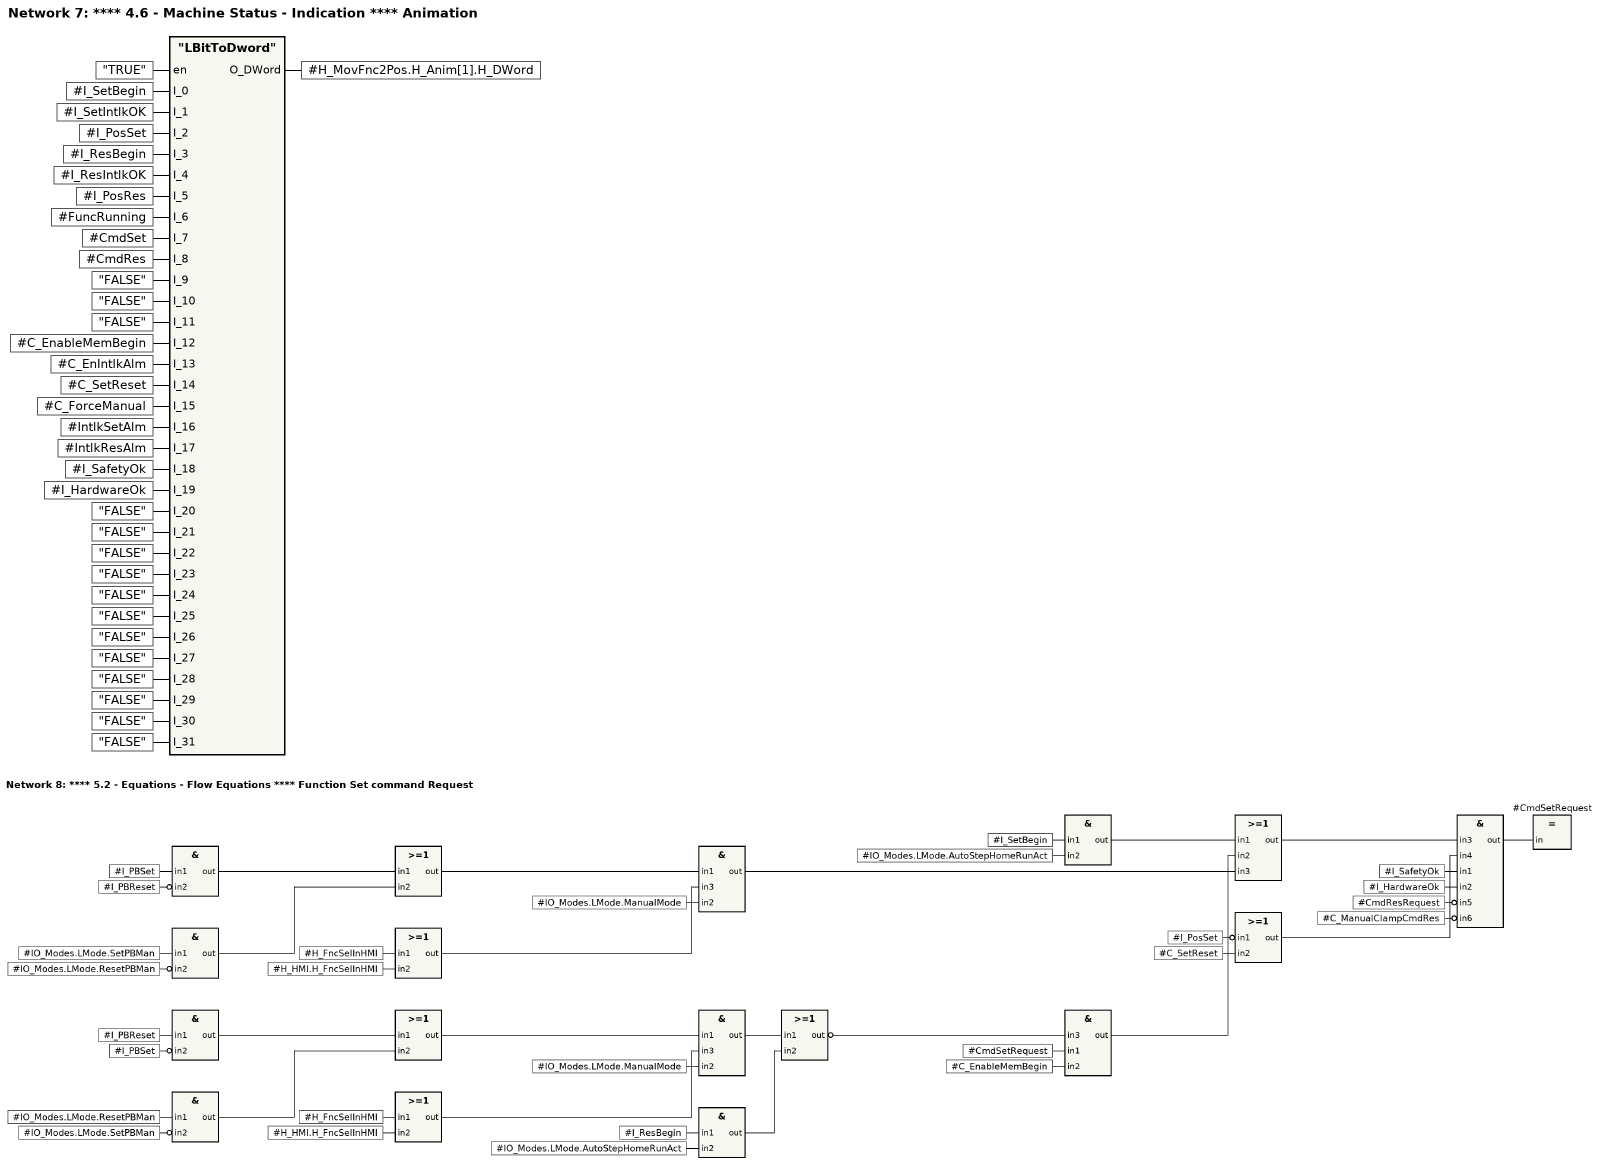
   IF "TRUE" THEN
       "LBitToDword"(I_0 := #I_SetBegin,
                     I_1 := #I_SetIntlkOK,
                     I_2 := #I_PosSet,
                     I_3 := #I_ResBegin,
                     I_4 := #I_ResIntlkOK,
                     I_5 := #I_PosRes,
                     I_6 := #FuncRunning,
                     I_7 := #CmdSet,
                     I_8 := #CmdRes,
                     I_9 := "FALSE",
                     I_10 := "FALSE",
                     I_11 := "FALSE",
                     I_12 := #C_EnableMemBegin,
                     I_13 := #C_EnIntlkAlm,
                     I_14 := #C_SetReset,
                     I_15 := #C_ForceManual,
                     I_16 := #IntlkSetAlm,
                     I_17 := #IntlkResAlm,
                     I_18 := #I_SafetyOk,
                     I_19 := #I_HardwareOk,
                     I_20 := "FALSE",
                     I_21 := "FALSE",
                     I_22 := "FALSE",
                     I_23 := "FALSE",
                     I_24 := "FALSE",
                     I_25 := "FALSE",
                     I_26 := "FALSE",
                     I_27 := "FALSE",
                     I_28 := "FALSE",
                     I_29 := "FALSE",
                     I_30 := "FALSE",
                     I_31 := "FALSE",
                     O_DWord => #H_MovFnc2Pos.H_Anim[1].H_DWord);
   END_IF;
END_REGION

REGION Network 8: **** 5.2 - Equations - Flow Equations **** Function Set command Request
   // Function Set command Request
   #CmdSetRequest := ((#I_SetBegin AND #IO_Modes.LMode.AutoStepHomeRunAct) OR (NOT ((((#I_PBReset AND NOT #I_PBSet) OR (#IO_Modes.LMode.ResetPBMan AND NOT #IO_Modes.LMode.SetPBMan)) AND (#H_FncSelInHMI OR #H_HMI.H_FncSelInHMI) AND #IO_Modes.LMode.ManualMode) OR (#I_ResBegin AND #IO_Modes.LMode.AutoStepHomeRunAct)) AND #CmdSetRequest AND #C_EnableMemBegin) OR (((#I_PBSet AND NOT #I_PBReset) OR (#IO_Modes.LMode.SetPBMan AND NOT #IO_Modes.LMode.ResetPBMan)) AND (#H_FncSelInHMI OR #H_HMI.H_FncSelInHMI) AND #IO_Modes.LMode.ManualMode)) AND (NOT #I_PosSet OR #C_SetReset) AND #I_SafetyOk AND #I_HardwareOk AND NOT #CmdResRequest AND NOT #C_ManualClampCmdRes;
END_REGION

REGION Network 9: **** 5.2 - Equations - Flow Equations **** Function Reset command Request
   // Function Reset command Request
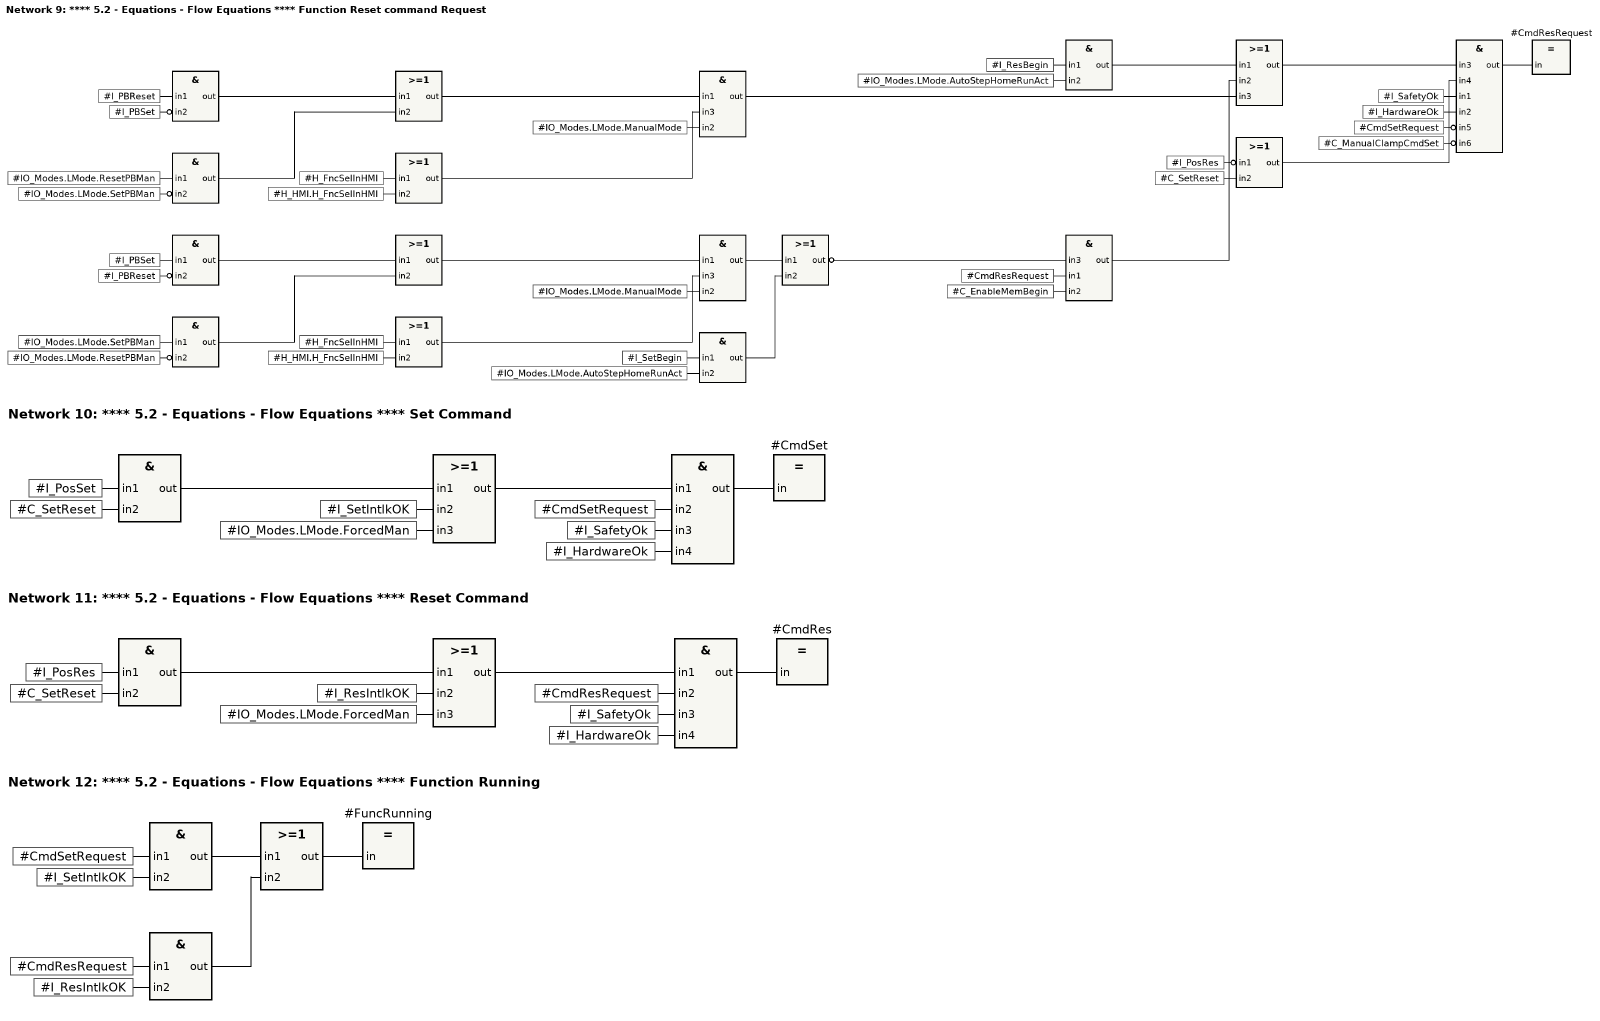
   #CmdResRequest := ((#I_ResBegin AND #IO_Modes.LMode.AutoStepHomeRunAct) OR (NOT ((((#I_PBSet AND NOT #I_PBReset) OR (#IO_Modes.LMode.SetPBMan AND NOT #IO_Modes.LMode.ResetPBMan)) AND (#H_FncSelInHMI OR #H_HMI.H_FncSelInHMI) AND #IO_Modes.LMode.ManualMode) OR (#I_SetBegin AND #IO_Modes.LMode.AutoStepHomeRunAct)) AND #CmdResRequest AND #C_EnableMemBegin) OR (((#I_PBReset AND NOT #I_PBSet) OR (#IO_Modes.LMode.ResetPBMan AND NOT #IO_Modes.LMode.SetPBMan)) AND (#H_FncSelInHMI OR #H_HMI.H_FncSelInHMI) AND #IO_Modes.LMode.ManualMode)) AND (NOT #I_PosRes OR #C_SetReset) AND #I_SafetyOk AND #I_HardwareOk AND NOT #CmdSetRequest AND NOT #C_ManualClampCmdSet;
END_REGION

REGION Network 10: **** 5.2 - Equations - Flow Equations **** Set Command
   // Set Command
   #CmdSet := ((#I_PosSet AND #C_SetReset) OR #I_SetIntlkOK OR #IO_Modes.LMode.ForcedMan) AND #CmdSetRequest AND #I_SafetyOk AND #I_HardwareOk;
END_REGION

REGION Network 11: **** 5.2 - Equations - Flow Equations **** Reset Command
   // Reset Command
   #CmdRes := ((#I_PosRes AND #C_SetReset) OR #I_ResIntlkOK OR #IO_Modes.LMode.ForcedMan) AND #CmdResRequest AND #I_SafetyOk AND #I_HardwareOk;
END_REGION

REGION Network 12: **** 5.2 - Equations - Flow Equations **** Function Running
   // Function Running
   #FuncRunning := (#CmdSetRequest AND #I_SetIntlkOK) OR (#CmdResRequest AND #I_ResIntlkOK);
END_REGION

REGION Network 13: **** 5.2 - Equations - Flow Equations **** Function Running Memory
   // Function Running Memory
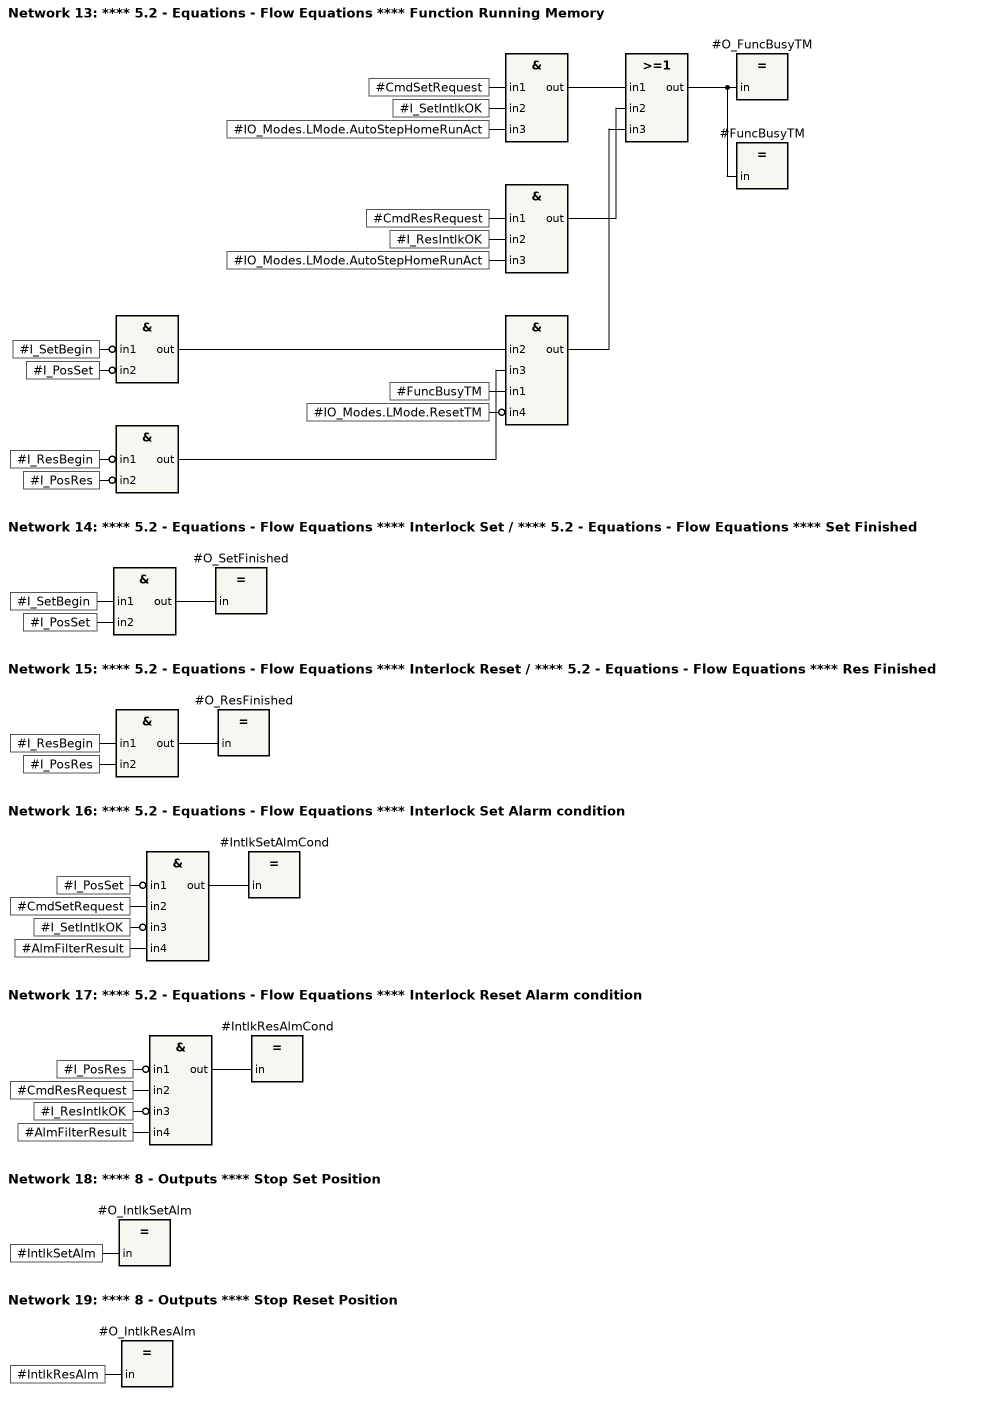
   #O_FuncBusyTM := (#CmdSetRequest AND #I_SetIntlkOK AND #IO_Modes.LMode.AutoStepHomeRunAct) OR (#CmdResRequest AND #I_ResIntlkOK AND #IO_Modes.LMode.AutoStepHomeRunAct) OR (NOT #I_SetBegin AND NOT #I_PosSet AND NOT #I_ResBegin AND NOT #I_PosRes AND #FuncBusyTM AND NOT #IO_Modes.LMode.ResetTM);
   #FuncBusyTM := #O_FuncBusyTM;
END_REGION

REGION Network 14: **** 5.2 - Equations - Flow Equations **** Interlock Set / **** 5.2 - Equations - Flow Equations **** Set Finished
   // Interlock Set
   #O_SetFinished := #I_SetBegin AND #I_PosSet;
END_REGION

REGION Network 15: **** 5.2 - Equations - Flow Equations **** Interlock Reset / **** 5.2 - Equations - Flow Equations **** Res Finished
   // Interlock Reset
   #O_ResFinished := #I_ResBegin AND #I_PosRes;
END_REGION

REGION Network 16: **** 5.2 - Equations - Flow Equations **** Interlock Set Alarm condition
   // Interlock Set Alarm condition
   #IntlkSetAlmCond := NOT #I_PosSet AND #CmdSetRequest AND NOT #I_SetIntlkOK AND #AlmFilterResult;
END_REGION

REGION Network 17: **** 5.2 - Equations - Flow Equations **** Interlock Reset Alarm condition
   // Interlock Reset Alarm condition
   #IntlkResAlmCond := NOT #I_PosRes AND #CmdResRequest AND NOT #I_ResIntlkOK AND #AlmFilterResult;
END_REGION

REGION Network 18: **** 8 - Outputs **** Stop Set Position
   // Stop Set Position
   #O_IntlkSetAlm := #IntlkSetAlm;
END_REGION

REGION Network 19: **** 8 - Outputs **** Stop Reset Position
   // Stop Reset Position
   #O_IntlkResAlm := #IntlkResAlm;
END_REGION

REGION Network 20: **** 8 - Outputs **** Function is Selected in manual Mode
   // Function is Selected in manual Mode
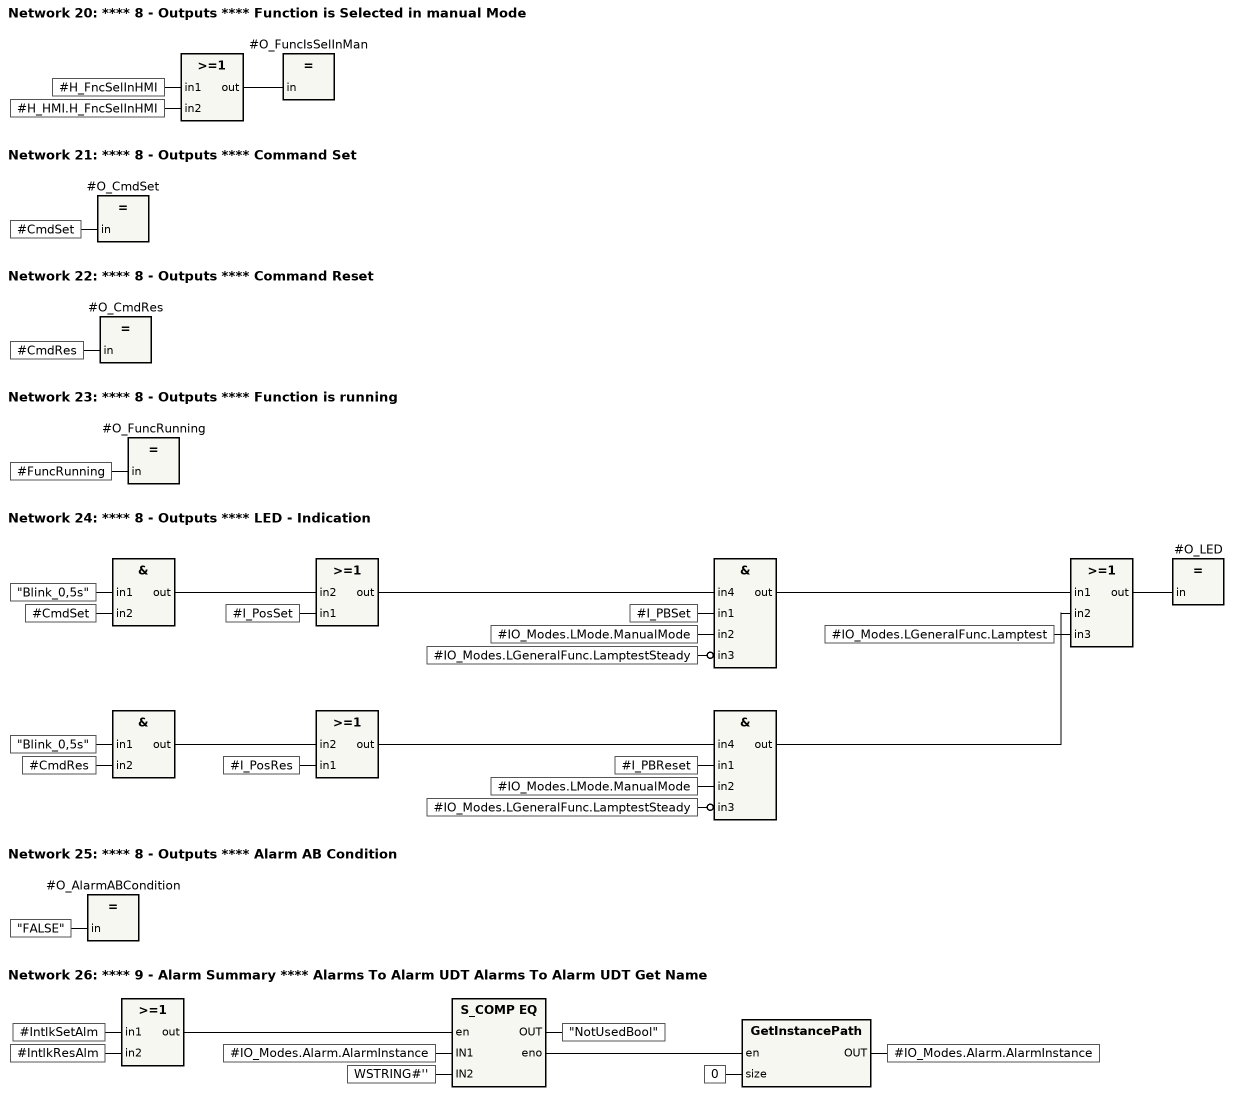
   #O_FuncIsSelInMan := #H_FncSelInHMI OR #H_HMI.H_FncSelInHMI;
END_REGION

REGION Network 21: **** 8 - Outputs **** Command Set
   // Command set
   #O_CmdSet := #CmdSet;
END_REGION

REGION Network 22: **** 8 - Outputs **** Command Reset
   // Command Reset
   #O_CmdRes := #CmdRes;
END_REGION

REGION Network 23: **** 8 - Outputs **** Function is running
   // Function is running
   #O_FuncRunning := #FuncRunning;
END_REGION

REGION Network 24: **** 8 - Outputs **** LED - Indication
   // LED - Indication
   #O_LED := ((("Blink_0,5s" AND #CmdSet) OR #I_PosSet) AND #I_PBSet AND #IO_Modes.LMode.ManualMode AND NOT #IO_Modes.LGeneralFunc.LamptestSteady) OR ((("Blink_0,5s" AND #CmdRes) OR #I_PosRes) AND #I_PBReset AND #IO_Modes.LMode.ManualMode AND NOT #IO_Modes.LGeneralFunc.LamptestSteady) OR #IO_Modes.LGeneralFunc.Lamptest;
END_REGION

REGION Network 25: **** 8 - Outputs **** Alarm AB Condition
   // Alarm AB Condition
   #O_AlarmABCondition := "FALSE";
END_REGION

REGION Network 26: **** 9 - Alarm Summary **** Alarms To Alarm UDT Alarms To Alarm UDT Get Name
   // Alarm / Alarm D
   S_COMP(EN := #IntlkSetAlm OR #IntlkResAlm,
          IN1 := #IO_Modes.Alarm.AlarmInstance,
          IN2 := WSTRING#'',
          OUT => "NotUsedBool",
          ENO => #_w1);
   IF #_w1 THEN GetInstancePath(size := 0, OUT => #IO_Modes.Alarm.AlarmInstance); END_IF;
END_REGION

REGION Network 27: **** 9 - Alarm Summary **** Alarms To Alarm UDT
   // Alarm / Alarm D
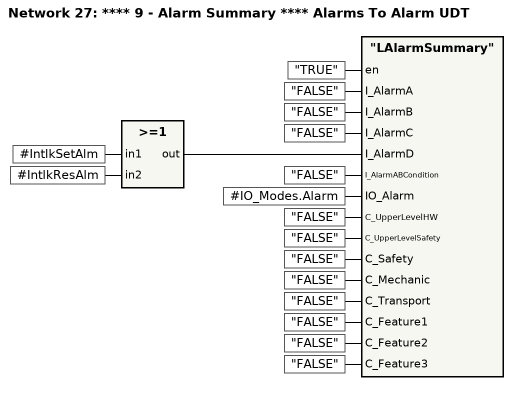
   IF "TRUE" THEN
       "LAlarmSummary"(I_AlarmA := "FALSE",
                       I_AlarmB := "FALSE",
                       I_AlarmC := "FALSE",
                       I_AlarmD := #IntlkSetAlm OR #IntlkResAlm,
                       I_AlarmABCondition := "FALSE",
                       IO_Alarm := #IO_Modes.Alarm,
                       C_UpperLevelHW := "FALSE",
                       C_UpperLevelSafety := "FALSE",
                       C_Safety := "FALSE",
                       C_Mechanic := "FALSE",
                       C_Transport := "FALSE",
                       C_Feature1 := "FALSE",
                       C_Feature2 := "FALSE",
                       C_Feature3 := "FALSE");
   END_IF;
END_REGION
END_FUNCTION_BLOCK

FUNCTION_BLOCK "LGeneralReverse"   // FB1103, FBD
TITLE = LGeneralReverse
{ S7_Optimized_Access := 'TRUE' }
VERSION : 0.1
// stored: AutoNumber false, IsIECCheckEnabled false, IsRetainMemResEnabled false, MemoryReserve 100, SetENOAutomatically False, UDAEnableTagReadback false
   VAR_INPUT
      I_GeneralReverseSw { ExternalAccessible := 'False'; ExternalVisible := 'False'; ExternalWritable := 'False'} : Bool;   // General reverse switch
      I_FbkContactorFwd { ExternalAccessible := 'False'; ExternalVisible := 'False'; ExternalWritable := 'False'} : Bool;   // Feedback contactor Forward
      I_FbkContactorBwd { ExternalAccessible := 'False'; ExternalVisible := 'False'; ExternalWritable := 'False'} : Bool;   // Feedback contactor Backward
      I_EnableAlarm { ExternalAccessible := 'False'; ExternalVisible := 'False'; ExternalWritable := 'False'} : Bool;   // Enable alarm / Enable Alarm
      I_ResetFbkAlarm { ExternalAccessible := 'False'; ExternalVisible := 'False'; ExternalWritable := 'False'} : Bool;   // Reset feedback alarm / Alarm reset pushbutton is activated
      C_FeedbackUsed { ExternalAccessible := 'False'; ExternalVisible := 'False'; ExternalWritable := 'False'} : Bool;   // Config Feedback used
   END_VAR
   VAR_OUTPUT
      O_ContactorFwd { ExternalAccessible := 'False'; ExternalVisible := 'False'; ExternalWritable := 'False'} : Bool;   // Activate low speed contactor / Activate Forward contactor
      O_ContactorBwd { ExternalAccessible := 'False'; ExternalVisible := 'False'; ExternalWritable := 'False'} : Bool;   // Activate High Speed contactor / Activate Backward contactor
      O_GenRevSw { ExternalAccessible := 'False'; ExternalVisible := 'False'; ExternalWritable := 'False'} : Bool;   // General reverse switch
      O_AlarmABCondition { ExternalAccessible := 'False'; ExternalVisible := 'False'; ExternalWritable := 'False'} : Bool;   // Alarm AB Condition
      O_AlarmA { ExternalAccessible := 'False'; ExternalVisible := 'False'; ExternalWritable := 'False'} : Bool;   // Alarm A
      O_AlarmB { ExternalAccessible := 'False'; ExternalVisible := 'False'; ExternalWritable := 'False'} : Bool;   // Alarm B
      O_AlarmC { ExternalAccessible := 'False'; ExternalVisible := 'False'; ExternalWritable := 'False'} : Bool;   // Alarm C
      O_AlarmD { ExternalAccessible := 'False'; ExternalVisible := 'False'; ExternalWritable := 'False'} : Bool;   // Alarm D
      H_AlarmDWord { ExternalAccessible := 'False'; ExternalVisible := 'False'; ExternalWritable := 'False'} : DWord;   // Alarm Word
   END_VAR
   VAR_IN_OUT
      IO_Modes : "Modes";   // Modes
      H_HMI : "H_HMI";   // Icon Animation
      H_GeneralReverse : "H_GeneralReverse";   // Animation
   END_VAR
   VAR
      AB_FbkContactorFwd { ExternalAccessible := 'False'; ExternalVisible := 'False'; ExternalWritable := 'False'} : Bool;   // Feedback error Contactor Forward
      AB_FbkContactorBwd { ExternalAccessible := 'False'; ExternalVisible := 'False'; ExternalWritable := 'False'} : Bool;   // Feedback error Contactor Backward
      AB_GeneralReverseSw { ExternalAccessible := 'False'; ExternalVisible := 'False'; ExternalWritable := 'False'} : Bool;   // General reverse is activated
      AC_GeneralReverseSw { ExternalAccessible := 'False'; ExternalVisible := 'False'; ExternalWritable := 'False'} : Bool;   // General reverse Switch is active
      FbkContactorFwdAlmCond { ExternalAccessible := 'False'; ExternalVisible := 'False'; ExternalWritable := 'False'} : Bool;   // Motor protection alarm condition / Motor protection Alarm condition / Feedback Contactor Forward Alarm condition
      FbkContactorBwdAlmCond { ExternalAccessible := 'False'; ExternalVisible := 'False'; ExternalWritable := 'False'} : Bool;   // Motor protection alarm condition / Motor protection Alarm condition / Feedback Contactor Backward Alarm condition
      AlarmA { ExternalAccessible := 'False'; ExternalVisible := 'False'; ExternalWritable := 'False'} : Bool;   // Alarm A
      AlarmB { ExternalAccessible := 'False'; ExternalVisible := 'False'; ExternalWritable := 'False'} : Bool;   // Alarm B
      AlarmC { ExternalAccessible := 'False'; ExternalVisible := 'False'; ExternalWritable := 'False'} : Bool;   // Alarm C
      AlarmD { ExternalAccessible := 'False'; ExternalVisible := 'False'; ExternalWritable := 'False'} : Bool;   // Alarm D
      AlarmABCondition { ExternalAccessible := 'False'; ExternalVisible := 'False'; ExternalWritable := 'False'} : Bool;   // Alarm AB Condition
      ContactorFwd { ExternalAccessible := 'False'; ExternalVisible := 'False'; ExternalWritable := 'False'} : Bool;   // Activate low speed contactor / Activate Forward contactor
      ContactorBwd { ExternalAccessible := 'False'; ExternalVisible := 'False'; ExternalWritable := 'False'} : Bool;   // Activate High Speed contactor / Activate Backward contactor
      _TimerInit { ExternalAccessible := 'False'; ExternalVisible := 'False'; ExternalWritable := 'False'} : TON_TIME;   // Timer
      _TimerContactorFwd { ExternalAccessible := 'False'; ExternalVisible := 'False'; ExternalWritable := 'False'} : TON_TIME;   // Timer
      _TimerContactorBwd { ExternalAccessible := 'False'; ExternalVisible := 'False'; ExternalWritable := 'False'} : TON_TIME;   // Timer
      _TimerContactorFwdFbk { ExternalAccessible := 'False'; ExternalVisible := 'False'; ExternalWritable := 'False'} : TON_TIME;   // Timer
      _TimerContactorBwdFbk { ExternalAccessible := 'False'; ExternalVisible := 'False'; ExternalWritable := 'False'} : TON_TIME;   // Timer
      _ContactorFwdFbk { ExternalAccessible := 'False'; ExternalVisible := 'False'; ExternalWritable := 'False'} : "L1AlarmMultiIn";   // FB
      _ContactorBwdFbk { ExternalAccessible := 'False'; ExternalVisible := 'False'; ExternalWritable := 'False'} : "L1AlarmMultiIn";   // FB
      Edge { ExternalAccessible := 'False'; ExternalVisible := 'False'; ExternalWritable := 'False'} : Array[1..10] of Bool;   // Edge
   END_VAR
   VAR_TEMP   // added for the SCL form of the ladder/FBD networks
      _w1 : Bool;
      _w2 : Bool;
   END_VAR
BEGIN

REGION Network 1: ****2.1 - Enable Alarms **** Enable Contactor Forward Feedback Alarm
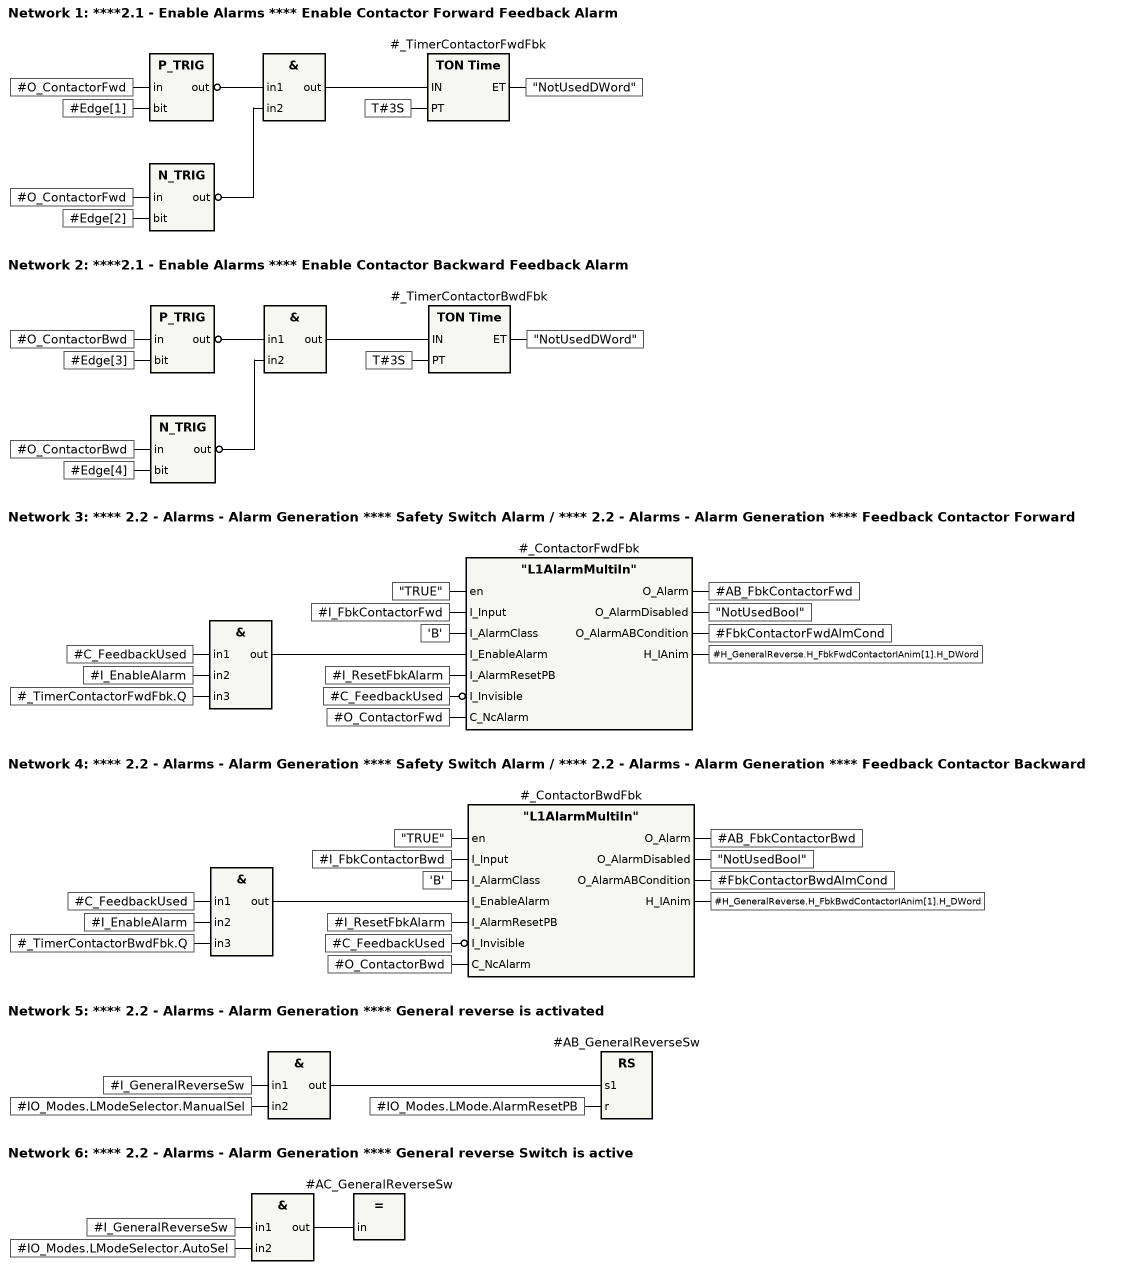
   #_w1 := #O_ContactorFwd AND NOT #Edge[1];   // rising edge
   #Edge[1] := #O_ContactorFwd;
   #_w2 := NOT #O_ContactorFwd AND #Edge[2];   // falling edge
   #Edge[2] := #O_ContactorFwd;
   #_TimerContactorFwdFbk(IN := NOT #_w1 AND NOT #_w2, PT := T#3S, ET => "NotUsedDWord");   // TON
END_REGION

REGION Network 2: ****2.1 - Enable Alarms **** Enable Contactor Backward Feedback Alarm
   #_w1 := #O_ContactorBwd AND NOT #Edge[3];   // rising edge
   #Edge[3] := #O_ContactorBwd;
   #_w2 := NOT #O_ContactorBwd AND #Edge[4];   // falling edge
   #Edge[4] := #O_ContactorBwd;
   #_TimerContactorBwdFbk(IN := NOT #_w1 AND NOT #_w2, PT := T#3S, ET => "NotUsedDWord");   // TON
END_REGION

REGION Network 3: **** 2.2 - Alarms - Alarm Generation **** Safety Switch Alarm / **** 2.2 - Alarms - Alarm Generation **** Feedback Contactor Forward
   // Safety Switch Alarm / Feedback error Contactor Forward
   IF "TRUE" THEN
       #_ContactorFwdFbk(I_Input := #I_FbkContactorFwd,   // "L1AlarmMultiIn"
                         I_AlarmClass := 'B',
                         I_EnableAlarm := #C_FeedbackUsed AND #I_EnableAlarm AND #_TimerContactorFwdFbk.Q,
                         I_AlarmResetPB := #I_ResetFbkAlarm,
                         I_Invisible := NOT #C_FeedbackUsed,
                         C_NcAlarm := #O_ContactorFwd,
                         O_Alarm => #AB_FbkContactorFwd,
                         O_AlarmDisabled => "NotUsedBool",
                         O_AlarmABCondition => #FbkContactorFwdAlmCond,
                         H_IAnim => #H_GeneralReverse.H_FbkFwdContactorIAnim[1].H_DWord);
   END_IF;
END_REGION

REGION Network 4: **** 2.2 - Alarms - Alarm Generation **** Safety Switch Alarm / **** 2.2 - Alarms - Alarm Generation **** Feedback Contactor Backward
   // Safety Switch Alarm / Feedback error Contactor Backward
   IF "TRUE" THEN
       #_ContactorBwdFbk(I_Input := #I_FbkContactorBwd,   // "L1AlarmMultiIn"
                         I_AlarmClass := 'B',
                         I_EnableAlarm := #C_FeedbackUsed AND #I_EnableAlarm AND #_TimerContactorBwdFbk.Q,
                         I_AlarmResetPB := #I_ResetFbkAlarm,
                         I_Invisible := NOT #C_FeedbackUsed,
                         C_NcAlarm := #O_ContactorBwd,
                         O_Alarm => #AB_FbkContactorBwd,
                         O_AlarmDisabled => "NotUsedBool",
                         O_AlarmABCondition => #FbkContactorBwdAlmCond,
                         H_IAnim => #H_GeneralReverse.H_FbkBwdContactorIAnim[1].H_DWord);
   END_IF;
END_REGION

REGION Network 5: **** 2.2 - Alarms - Alarm Generation **** General reverse is activated
   IF #IO_Modes.LMode.AlarmResetPB THEN
       #AB_GeneralReverseSw := FALSE;   // RS flip-flop
   END_IF;
   IF #I_GeneralReverseSw AND #IO_Modes.LModeSelector.ManualSel THEN #AB_GeneralReverseSw := TRUE; END_IF;
END_REGION

REGION Network 6: **** 2.2 - Alarms - Alarm Generation **** General reverse Switch is active
   #AC_GeneralReverseSw := #I_GeneralReverseSw AND #IO_Modes.LModeSelector.AutoSel;
END_REGION

REGION Network 7: **** 4.6 - Machine Status - Indication **** Low Speed Contactor Animation / **** 4.6 - Machine Status - Indication **** Forward Contactor Animation
   // Low speed Contactor Animation
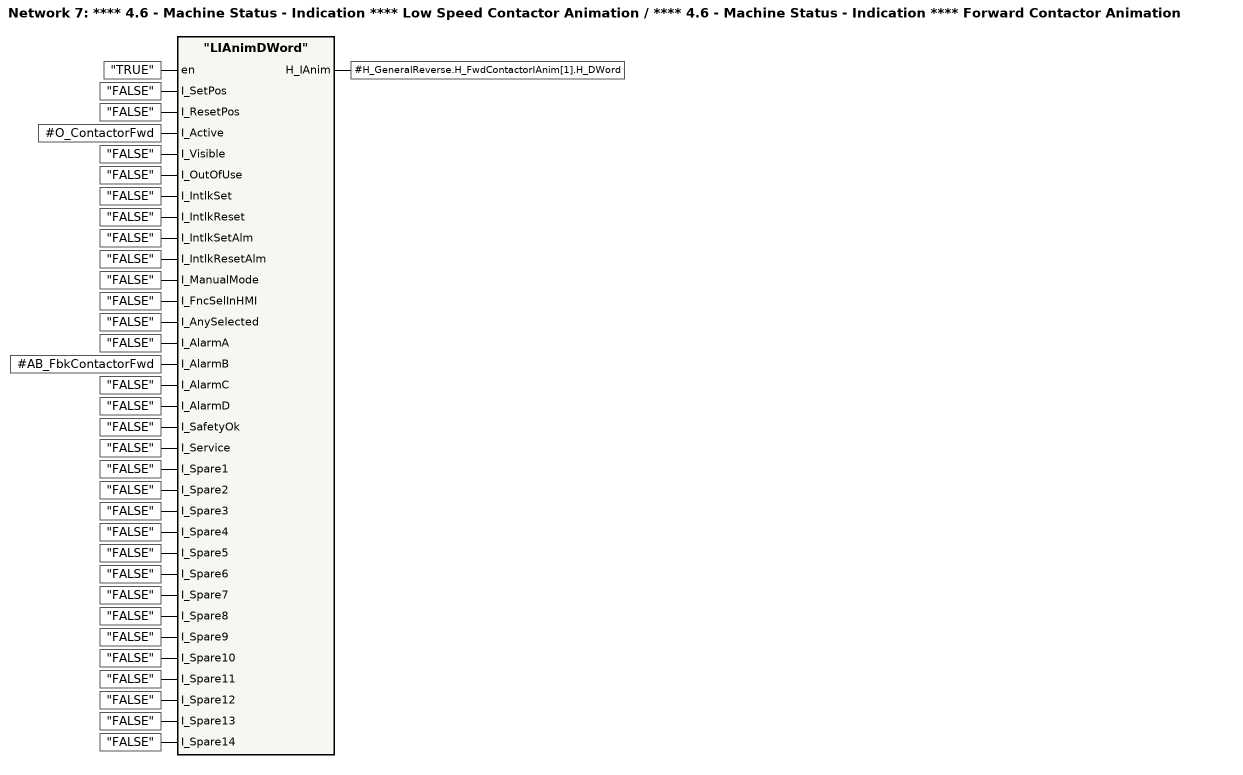
   IF "TRUE" THEN
       "LIAnimDWord"(I_SetPos := "FALSE",
                     I_ResetPos := "FALSE",
                     I_Active := #O_ContactorFwd,
                     I_Visible := "FALSE",
                     I_OutOfUse := "FALSE",
                     I_IntlkSet := "FALSE",
                     I_IntlkReset := "FALSE",
                     I_IntlkSetAlm := "FALSE",
                     I_IntlkResetAlm := "FALSE",
                     I_ManualMode := "FALSE",
                     I_FncSelInHMI := "FALSE",
                     I_AnySelected := "FALSE",
                     I_AlarmA := "FALSE",
                     I_AlarmB := #AB_FbkContactorFwd,
                     I_AlarmC := "FALSE",
                     I_AlarmD := "FALSE",
                     I_SafetyOk := "FALSE",
                     I_Service := "FALSE",
                     I_Spare1 := "FALSE",
                     I_Spare2 := "FALSE",
                     I_Spare3 := "FALSE",
                     I_Spare4 := "FALSE",
                     I_Spare5 := "FALSE",
                     I_Spare6 := "FALSE",
                     I_Spare7 := "FALSE",
                     I_Spare8 := "FALSE",
                     I_Spare9 := "FALSE",
                     I_Spare10 := "FALSE",
                     I_Spare11 := "FALSE",
                     I_Spare12 := "FALSE",
                     I_Spare13 := "FALSE",
                     I_Spare14 := "FALSE",
                     H_IAnim => #H_GeneralReverse.H_FwdContactorIAnim[1].H_DWord);
   END_IF;
END_REGION

REGION Network 8: **** 4.6 - Machine Status - Indication **** High Speed Contactor Animation / **** 4.6 - Machine Status - Indication **** Backward Contactor Animation
   // High Speed Contactor Animation
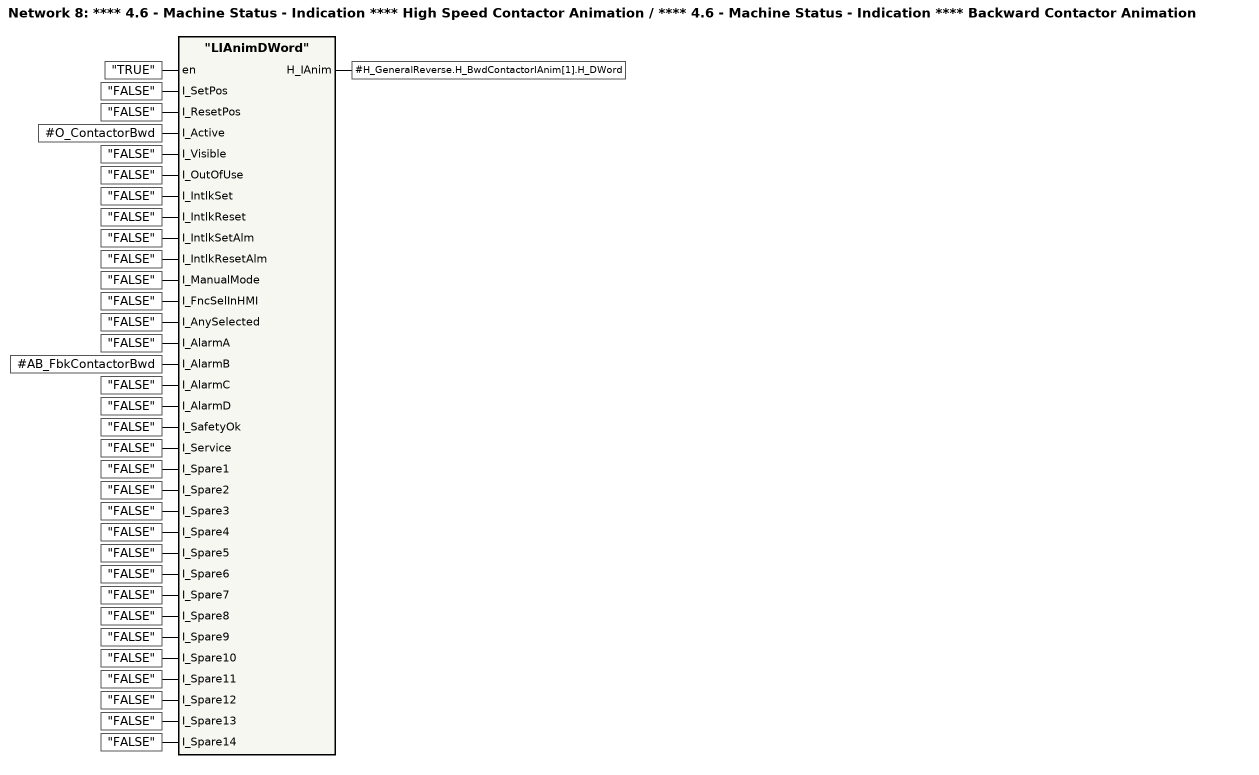
   IF "TRUE" THEN
       "LIAnimDWord"(I_SetPos := "FALSE",
                     I_ResetPos := "FALSE",
                     I_Active := #O_ContactorBwd,
                     I_Visible := "FALSE",
                     I_OutOfUse := "FALSE",
                     I_IntlkSet := "FALSE",
                     I_IntlkReset := "FALSE",
                     I_IntlkSetAlm := "FALSE",
                     I_IntlkResetAlm := "FALSE",
                     I_ManualMode := "FALSE",
                     I_FncSelInHMI := "FALSE",
                     I_AnySelected := "FALSE",
                     I_AlarmA := "FALSE",
                     I_AlarmB := #AB_FbkContactorBwd,
                     I_AlarmC := "FALSE",
                     I_AlarmD := "FALSE",
                     I_SafetyOk := "FALSE",
                     I_Service := "FALSE",
                     I_Spare1 := "FALSE",
                     I_Spare2 := "FALSE",
                     I_Spare3 := "FALSE",
                     I_Spare4 := "FALSE",
                     I_Spare5 := "FALSE",
                     I_Spare6 := "FALSE",
                     I_Spare7 := "FALSE",
                     I_Spare8 := "FALSE",
                     I_Spare9 := "FALSE",
                     I_Spare10 := "FALSE",
                     I_Spare11 := "FALSE",
                     I_Spare12 := "FALSE",
                     I_Spare13 := "FALSE",
                     I_Spare14 := "FALSE",
                     H_IAnim => #H_GeneralReverse.H_BwdContactorIAnim[1].H_DWord);
   END_IF;
END_REGION

REGION Network 9: **** 4.6 - Machine Status - Indication **** Stop Detection Reset / **** 4.6 - Machine Status - Indications **** General Reverse Switch Animation
   // Stop Detection Reset
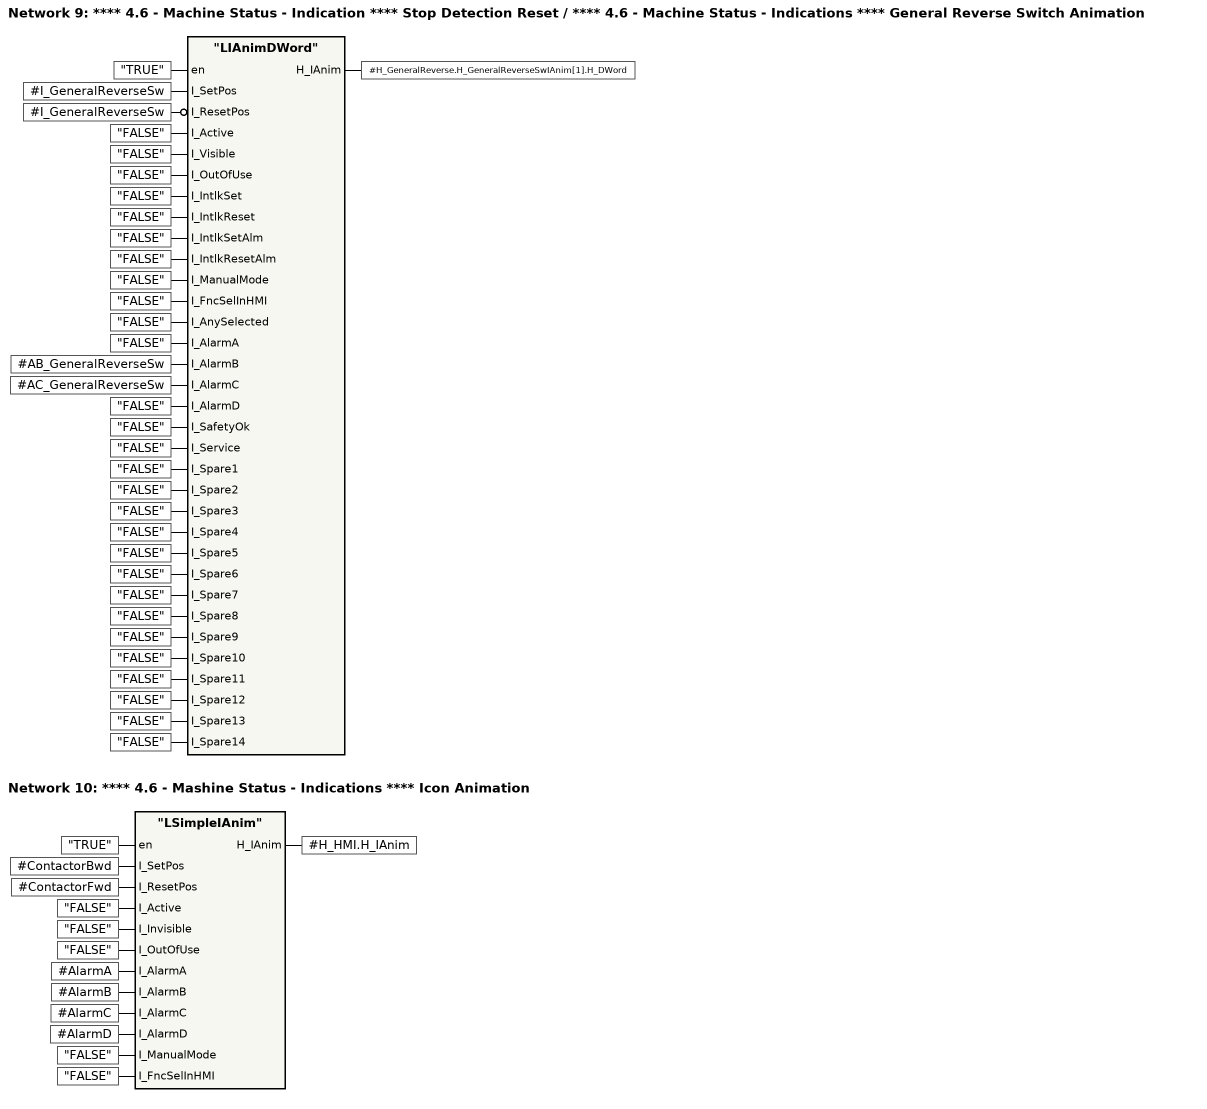
   IF "TRUE" THEN
       "LIAnimDWord"(I_SetPos := #I_GeneralReverseSw,
                     I_ResetPos := NOT #I_GeneralReverseSw,
                     I_Active := "FALSE",
                     I_Visible := "FALSE",
                     I_OutOfUse := "FALSE",
                     I_IntlkSet := "FALSE",
                     I_IntlkReset := "FALSE",
                     I_IntlkSetAlm := "FALSE",
                     I_IntlkResetAlm := "FALSE",
                     I_ManualMode := "FALSE",
                     I_FncSelInHMI := "FALSE",
                     I_AnySelected := "FALSE",
                     I_AlarmA := "FALSE",
                     I_AlarmB := #AB_GeneralReverseSw,
                     I_AlarmC := #AC_GeneralReverseSw,
                     I_AlarmD := "FALSE",
                     I_SafetyOk := "FALSE",
                     I_Service := "FALSE",
                     I_Spare1 := "FALSE",
                     I_Spare2 := "FALSE",
                     I_Spare3 := "FALSE",
                     I_Spare4 := "FALSE",
                     I_Spare5 := "FALSE",
                     I_Spare6 := "FALSE",
                     I_Spare7 := "FALSE",
                     I_Spare8 := "FALSE",
                     I_Spare9 := "FALSE",
                     I_Spare10 := "FALSE",
                     I_Spare11 := "FALSE",
                     I_Spare12 := "FALSE",
                     I_Spare13 := "FALSE",
                     I_Spare14 := "FALSE",
                     H_IAnim => #H_GeneralReverse.H_GeneralReverseSwIAnim[1].H_DWord);
   END_IF;
END_REGION

REGION Network 10: **** 4.6 - Mashine Status - Indications **** Icon Animation
   // Icon Animation
   IF "TRUE" THEN
       "LSimpleIAnim"(I_SetPos := #ContactorBwd,
                      I_ResetPos := #ContactorFwd,
                      I_Active := "FALSE",
                      I_Invisible := "FALSE",
                      I_OutOfUse := "FALSE",
                      I_AlarmA := #AlarmA,
                      I_AlarmB := #AlarmB,
                      I_AlarmC := #AlarmC,
                      I_AlarmD := #AlarmD,
                      I_ManualMode := "FALSE",
                      I_FncSelInHMI := "FALSE",
                      H_IAnim => #H_HMI.H_IAnim);
   END_IF;
END_REGION

REGION Network 11: **** 4.6 - Machine status - Indications **** Animation
   // Animation Word 1
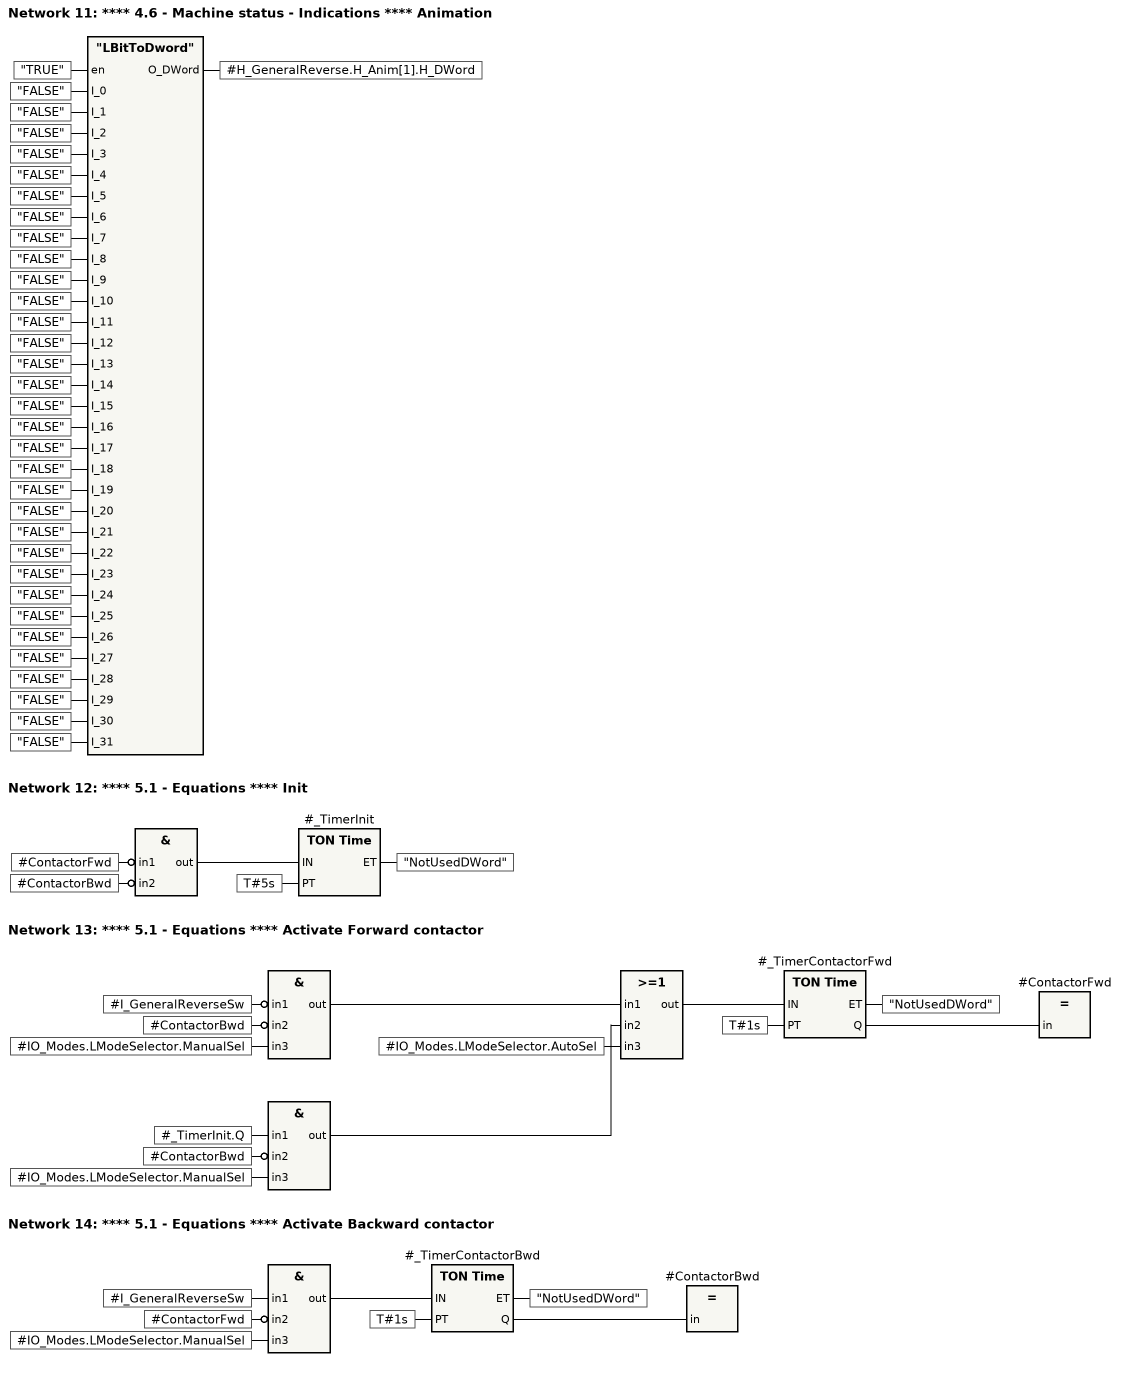
   IF "TRUE" THEN
       "LBitToDword"(I_0 := "FALSE",
                     I_1 := "FALSE",
                     I_2 := "FALSE",
                     I_3 := "FALSE",
                     I_4 := "FALSE",
                     I_5 := "FALSE",
                     I_6 := "FALSE",
                     I_7 := "FALSE",
                     I_8 := "FALSE",
                     I_9 := "FALSE",
                     I_10 := "FALSE",
                     I_11 := "FALSE",
                     I_12 := "FALSE",
                     I_13 := "FALSE",
                     I_14 := "FALSE",
                     I_15 := "FALSE",
                     I_16 := "FALSE",
                     I_17 := "FALSE",
                     I_18 := "FALSE",
                     I_19 := "FALSE",
                     I_20 := "FALSE",
                     I_21 := "FALSE",
                     I_22 := "FALSE",
                     I_23 := "FALSE",
                     I_24 := "FALSE",
                     I_25 := "FALSE",
                     I_26 := "FALSE",
                     I_27 := "FALSE",
                     I_28 := "FALSE",
                     I_29 := "FALSE",
                     I_30 := "FALSE",
                     I_31 := "FALSE",
                     O_DWord => #H_GeneralReverse.H_Anim[1].H_DWord);
   END_IF;
END_REGION

REGION Network 12: **** 5.1 - Equations **** Init
   #_TimerInit(IN := NOT #ContactorFwd AND NOT #ContactorBwd, PT := T#5s, ET => "NotUsedDWord");   // TON
END_REGION

REGION Network 13: **** 5.1 - Equations **** Activate Forward contactor
   #_TimerContactorFwd(IN := (NOT #I_GeneralReverseSw AND NOT #ContactorBwd AND #IO_Modes.LModeSelector.ManualSel) OR (#_TimerInit.Q AND NOT #ContactorBwd AND #IO_Modes.LModeSelector.ManualSel) OR #IO_Modes.LModeSelector.AutoSel,   // TON
                       PT := T#1s,
                       ET => "NotUsedDWord");
   #ContactorFwd := #_TimerContactorFwd.Q;
END_REGION

REGION Network 14: **** 5.1 - Equations **** Activate Backward contactor
   #_TimerContactorBwd(IN := #I_GeneralReverseSw AND NOT #ContactorFwd AND #IO_Modes.LModeSelector.ManualSel,   // TON
                       PT := T#1s,
                       ET => "NotUsedDWord");
   #ContactorBwd := #_TimerContactorBwd.Q;
END_REGION

REGION Network 15: **** 8 - Outputs **** Alarm AB Condition
   // Alarm AB Condition
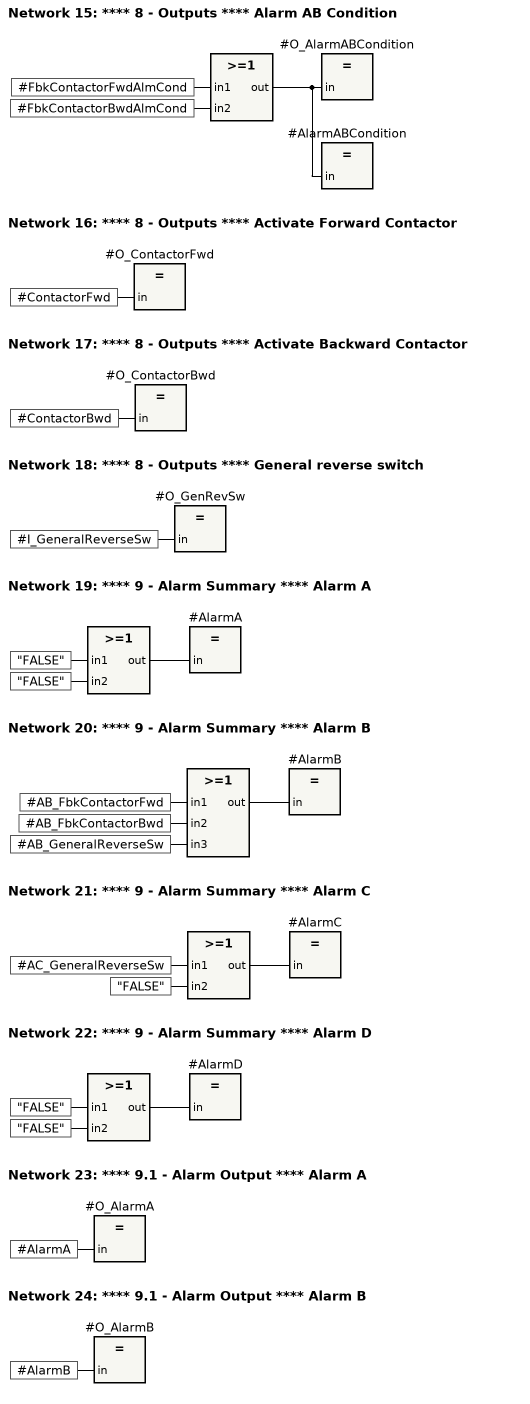
   #O_AlarmABCondition := #FbkContactorFwdAlmCond OR #FbkContactorBwdAlmCond;
   #AlarmABCondition := #O_AlarmABCondition;
END_REGION

REGION Network 16: **** 8 - Outputs **** Activate Forward Contactor
   #O_ContactorFwd := #ContactorFwd;
END_REGION

REGION Network 17: **** 8 - Outputs **** Activate Backward Contactor
   #O_ContactorBwd := #ContactorBwd;
END_REGION

REGION Network 18: **** 8 - Outputs **** General reverse switch
   #O_GenRevSw := #I_GeneralReverseSw;
END_REGION

REGION Network 19: **** 9 - Alarm Summary **** Alarm A
   // Alarm A
   #AlarmA := "FALSE" OR "FALSE";
END_REGION

REGION Network 20: **** 9 - Alarm Summary **** Alarm B
   // Alarm B
   #AlarmB := #AB_FbkContactorFwd OR #AB_FbkContactorBwd OR #AB_GeneralReverseSw;
END_REGION

REGION Network 21: **** 9 - Alarm Summary **** Alarm C
   // Alarm C
   #AlarmC := #AC_GeneralReverseSw OR "FALSE";
END_REGION

REGION Network 22: **** 9 - Alarm Summary **** Alarm D
   // Alarm D
   #AlarmD := "FALSE" OR "FALSE";
END_REGION

REGION Network 23: **** 9.1 - Alarm Output **** Alarm A
   // Alarm A
   #O_AlarmA := #AlarmA;
END_REGION

REGION Network 24: **** 9.1 - Alarm Output **** Alarm B
   // Alarm B
   #O_AlarmB := #AlarmB;
END_REGION

REGION Network 25: **** 9.1 - Alarm Output **** Alarm C
   // Alarm C
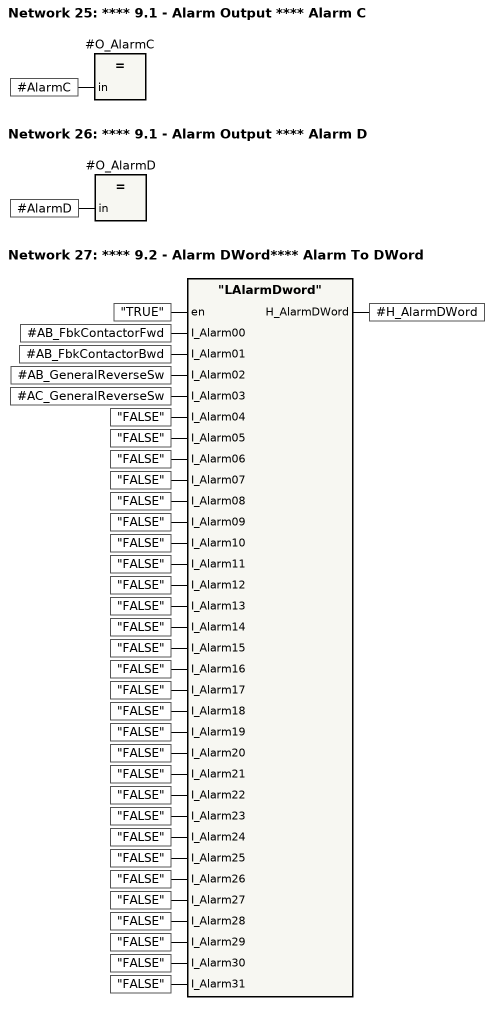
   #O_AlarmC := #AlarmC;
END_REGION

REGION Network 26: **** 9.1 - Alarm Output **** Alarm D
   // Alarm D
   #O_AlarmD := #AlarmD;
END_REGION

REGION Network 27: **** 9.2 - Alarm DWord**** Alarm To DWord
   // Alarm To DWord
   IF "TRUE" THEN
       "LAlarmDword"(I_Alarm00 := #AB_FbkContactorFwd,
                     I_Alarm01 := #AB_FbkContactorBwd,
                     I_Alarm02 := #AB_GeneralReverseSw,
                     I_Alarm03 := #AC_GeneralReverseSw,
                     I_Alarm04 := "FALSE",
                     I_Alarm05 := "FALSE",
                     I_Alarm06 := "FALSE",
                     I_Alarm07 := "FALSE",
                     I_Alarm08 := "FALSE",
                     I_Alarm09 := "FALSE",
                     I_Alarm10 := "FALSE",
                     I_Alarm11 := "FALSE",
                     I_Alarm12 := "FALSE",
                     I_Alarm13 := "FALSE",
                     I_Alarm14 := "FALSE",
                     I_Alarm15 := "FALSE",
                     I_Alarm16 := "FALSE",
                     I_Alarm17 := "FALSE",
                     I_Alarm18 := "FALSE",
                     I_Alarm19 := "FALSE",
                     I_Alarm20 := "FALSE",
                     I_Alarm21 := "FALSE",
                     I_Alarm22 := "FALSE",
                     I_Alarm23 := "FALSE",
                     I_Alarm24 := "FALSE",
                     I_Alarm25 := "FALSE",
                     I_Alarm26 := "FALSE",
                     I_Alarm27 := "FALSE",
                     I_Alarm28 := "FALSE",
                     I_Alarm29 := "FALSE",
                     I_Alarm30 := "FALSE",
                     I_Alarm31 := "FALSE",
                     H_AlarmDWord => #H_AlarmDWord);
   END_IF;
END_REGION
END_FUNCTION_BLOCK

FUNCTION_BLOCK "L1AlarmMultiIn"   // FB1426, FBD
TITLE = L1AlarmMultiIn
{ S7_Optimized_Access := 'FALSE' }
AUTHOR : VCC
FAMILY : AlarmHnd
NAME : 1Alarm
VERSION : 1.0
// ================================================================================
// This module is used inside another FB where one alarm shall be generated when 
// one (security) input becomes True.
// The alarm can be True only when the input Enable Alarm is also True.
// The alarm can be True only when the input Disable Alarm is False. When the 
// alarm is disabled from HMI, a boolean output is available to inform the upper 
// level and do action in the Alarm summary.
// When the conditions to generate the alarm disappear, a boolean output is 
// available to inform the upper level that the alarm can be reset.
// The alarm is reset by means of the AlarmResetPB signal.
// ================================================================================
// stored: AutoNumber false, IsIECCheckEnabled false, SetENOAutomatically False, UDAEnableTagReadback false
   VAR_INPUT
      I_Input { ExternalAccessible := 'False'; ExternalVisible := 'False'; ExternalWritable := 'False'} : Bool;   // Input signal of the alarm
      I_AlarmClass { ExternalAccessible := 'False'; ExternalVisible := 'False'; ExternalWritable := 'False'} : Char;   // Alarm class -> A - B - C - D or E
      I_EnableAlarm { ExternalAccessible := 'False'; ExternalVisible := 'False'; ExternalWritable := 'False'} : Bool := TRUE;   // Enable alarm from upper level
      I_AlarmResetPB { ExternalAccessible := 'False'; ExternalVisible := 'False'; ExternalWritable := 'False'} : Bool;   // Alarm reset pushbutton is activated
      I_Invisible { ExternalAccessible := 'False'; ExternalVisible := 'False'; ExternalWritable := 'False'} : Bool;   // Invisible
      C_NcAlarm { ExternalAccessible := 'False'; ExternalVisible := 'False'; ExternalWritable := 'False'} : Bool;   // Alarm contact NC
   END_VAR
   VAR_OUTPUT
      O_Alarm { ExternalAccessible := 'False'; ExternalVisible := 'False'; ExternalWritable := 'False'} : Bool;   // Alarm
      O_AlarmDisabled { ExternalAccessible := 'False'; ExternalVisible := 'False'; ExternalWritable := 'False'} : Bool;   // Alarm disabled from HMI
      O_AlarmABCondition { ExternalAccessible := 'False'; ExternalVisible := 'False'; ExternalWritable := 'False'} : Bool;   // Alarm AB condition
      H_IAnim { ExternalAccessible := 'False'; ExternalVisible := 'False'; ExternalWritable := 'False'} : DWord;
   END_VAR
   VAR DB_SPECIFIC
      H_In : Struct   // HMI
         DisableAlarm : Bool;   // Disable alarm from HMI
      END_STRUCT;
      H_Out : Struct   // HMI
         DBnr : Int;   // HMI Animation DB number
      END_STRUCT;
      Alarm { ExternalAccessible := 'False'; ExternalVisible := 'False'; ExternalWritable := 'False'} : Bool;   // Alarm
      AlarmClass_A { ExternalAccessible := 'False'; ExternalVisible := 'False'; ExternalWritable := 'False'} : Bool;   // The alarm is from alarm class A
      AlarmClass_B { ExternalAccessible := 'False'; ExternalVisible := 'False'; ExternalWritable := 'False'} : Bool;   // The alarm is from alarm class B
      AlarmClass_C { ExternalAccessible := 'False'; ExternalVisible := 'False'; ExternalWritable := 'False'} : Bool;   // The alarm is from alarm class C
      AlarmClass_D { ExternalAccessible := 'False'; ExternalVisible := 'False'; ExternalWritable := 'False'} : Bool;   // The alarm is from alarm class D
      AlarmClass_E { ExternalAccessible := 'False'; ExternalVisible := 'False'; ExternalWritable := 'False'} : Bool;   // The alarm is from alarm class E
      AlarmCond { ExternalAccessible := 'False'; ExternalVisible := 'False'; ExternalWritable := 'False'} : Bool;   // Alarm condition
      DBnr { ExternalAccessible := 'False'; ExternalVisible := 'False'; ExternalWritable := 'False'} : Int;   // HMI DB number
   END_VAR
BEGIN

NETWORK
TITLE = **** 1 - Inputs **** DB number
// DB number
      L     DINO;
      T     #DBnr;

NETWORK
TITLE = **** 1 - Inputs **** Alarm class
// Alarm class
// Alarm class = E
      L     #I_AlarmClass;
      L     'E';
      ==I;
      =     #AlarmClass_E;

// Alarm class = D
      L     #I_AlarmClass;
      L     'D';
      ==I;
      =     #AlarmClass_D;

// Alarm class = C
      L     #I_AlarmClass;
      L     'C';
      ==I;
      =     #AlarmClass_C;

// Alarm class = B
      L     #I_AlarmClass;
      L     'B';
      ==I;
      =     #AlarmClass_B;

// Alarm class = A
      AN    #AlarmClass_B;
      AN    #AlarmClass_C;
      AN    #AlarmClass_D;
      AN    #AlarmClass_E;
      =     #AlarmClass_A;


REGION Network 3: **** 2.2 - Alarms - Alarms Generation **** Alarm Condition
   // Condition for the Alarm
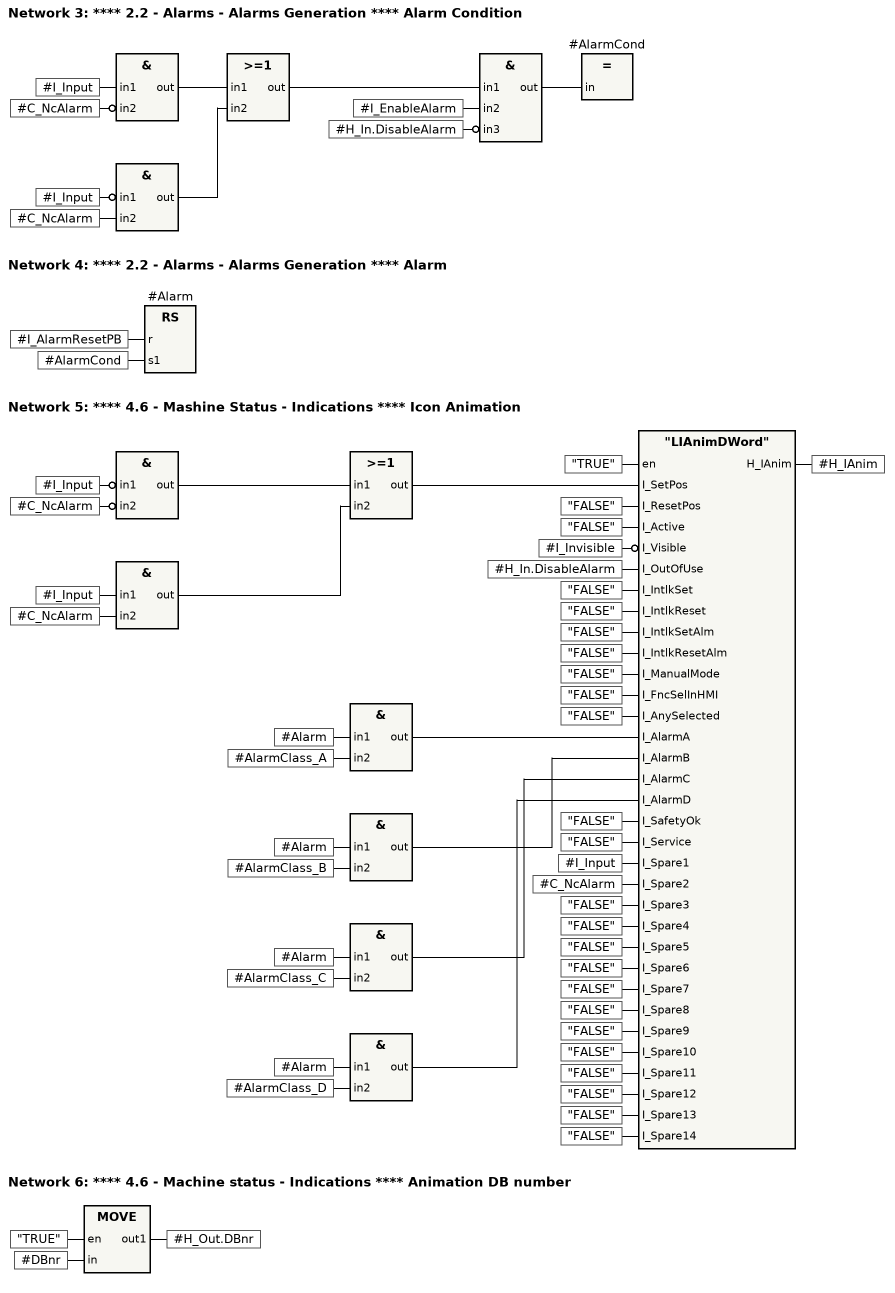
   #AlarmCond := ((#I_Input AND NOT #C_NcAlarm) OR (NOT #I_Input AND #C_NcAlarm)) AND #I_EnableAlarm AND NOT #H_In.DisableAlarm;
END_REGION

REGION Network 4: **** 2.2 - Alarms - Alarms Generation **** Alarm
   // Creation of the Alarm
   IF #I_AlarmResetPB THEN
       #Alarm := FALSE;   // RS flip-flop
   END_IF;
   IF #AlarmCond THEN #Alarm := TRUE; END_IF;
END_REGION

REGION Network 5: **** 4.6 - Mashine Status - Indications **** Icon Animation
   // Icon Animation
   IF "TRUE" THEN
       "LIAnimDWord"(I_SetPos := (NOT #I_Input AND NOT #C_NcAlarm) OR (#I_Input AND #C_NcAlarm),
                     I_ResetPos := "FALSE",
                     I_Active := "FALSE",
                     I_Visible := NOT #I_Invisible,
                     I_OutOfUse := #H_In.DisableAlarm,
                     I_IntlkSet := "FALSE",
                     I_IntlkReset := "FALSE",
                     I_IntlkSetAlm := "FALSE",
                     I_IntlkResetAlm := "FALSE",
                     I_ManualMode := "FALSE",
                     I_FncSelInHMI := "FALSE",
                     I_AnySelected := "FALSE",
                     I_AlarmA := #Alarm AND #AlarmClass_A,
                     I_AlarmB := #Alarm AND #AlarmClass_B,
                     I_AlarmC := #Alarm AND #AlarmClass_C,
                     I_AlarmD := #Alarm AND #AlarmClass_D,
                     I_SafetyOk := "FALSE",
                     I_Service := "FALSE",
                     I_Spare1 := #I_Input,
                     I_Spare2 := #C_NcAlarm,
                     I_Spare3 := "FALSE",
                     I_Spare4 := "FALSE",
                     I_Spare5 := "FALSE",
                     I_Spare6 := "FALSE",
                     I_Spare7 := "FALSE",
                     I_Spare8 := "FALSE",
                     I_Spare9 := "FALSE",
                     I_Spare10 := "FALSE",
                     I_Spare11 := "FALSE",
                     I_Spare12 := "FALSE",
                     I_Spare13 := "FALSE",
                     I_Spare14 := "FALSE",
                     H_IAnim => #H_IAnim);
   END_IF;
END_REGION

REGION Network 6: **** 4.6 - Machine status - Indications **** Animation DB number
   IF "TRUE" THEN #H_Out.DBnr := #DBnr; END_IF;
END_REGION

REGION Network 7: *** 8 - Outputs **** Disable alarm
   // Alarm disabled from HMI
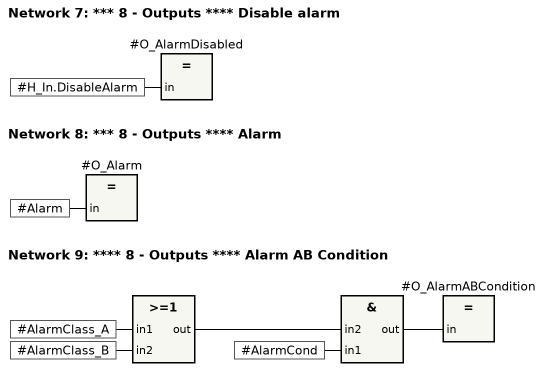
   #O_AlarmDisabled := #H_In.DisableAlarm;
END_REGION

REGION Network 8: *** 8 - Outputs **** Alarm
   // Output of the Alarm
   #O_Alarm := #Alarm;
END_REGION

REGION Network 9: **** 8 - Outputs **** Alarm AB Condition
   // Alarm Resetable
   #O_AlarmABCondition := (#AlarmClass_A OR #AlarmClass_B) AND #AlarmCond;
END_REGION
END_FUNCTION_BLOCK

FUNCTION_BLOCK "L1SignalHmi"   // FB1106, FBD
TITLE = L1SignalHmi
{ S7_Optimized_Access := 'FALSE' }
AUTHOR : VCT
FAMILY : VCT
NAME : L1SigHMI
VERSION : 1.0
// ===============================================================================
// This module handles the HMI functions for one signal
// ===============================================================================
// stored: AutoNumber false, IsIECCheckEnabled false, SetENOAutomatically False, UDAEnableTagReadback false
   VAR_INPUT
      I_Signal { ExternalAccessible := 'False'; ExternalVisible := 'False'; ExternalWritable := 'False'} : Bool;   // The signal
      I_SignalCheckOn { ExternalAccessible := 'False'; ExternalVisible := 'False'; ExternalWritable := 'False'} : Bool;   // Check signal is on
      I_SignalCheckOff { ExternalAccessible := 'False'; ExternalVisible := 'False'; ExternalWritable := 'False'} : Bool;   // Check signal is off
      I_EnableAlarm { ExternalAccessible := 'False'; ExternalVisible := 'False'; ExternalWritable := 'False'} : Bool;   // Enable alarms
      I_AlarmResetPB { ExternalAccessible := 'False'; ExternalVisible := 'False'; ExternalWritable := 'False'} : Bool;   // Alarm reset pushbutton is activated
   END_VAR
   VAR_OUTPUT
      O_SignalOn { ExternalAccessible := 'False'; ExternalVisible := 'False'; ExternalWritable := 'False'} : Bool;   // Detection signal to use in program
      O_SignalAlmReqOn { ExternalAccessible := 'False'; ExternalVisible := 'False'; ExternalWritable := 'False'} : Bool;   // Request on alarm
      O_SignalAlmReqOff { ExternalAccessible := 'False'; ExternalVisible := 'False'; ExternalWritable := 'False'} : Bool;   // Request off alarm
      O_AlarmABCondition { ExternalAccessible := 'False'; ExternalVisible := 'False'; ExternalWritable := 'False'} : Bool;   // Alarm AB condition
      H_IAnim { ExternalAccessible := 'False'; ExternalVisible := 'False'; ExternalWritable := 'False'} : Word;   // For animation of the icon
   END_VAR
   VAR DB_SPECIFIC
      H_Out : Struct   // HMI
         Anim : Word;   // HMI Animation of the object
      END_STRUCT;
      SignalCheckOnAlarm { ExternalAccessible := 'False'; ExternalVisible := 'False'; ExternalWritable := 'False'} : Bool;   // Detection is not on
      SignalCheckOffAlarm { ExternalAccessible := 'False'; ExternalVisible := 'False'; ExternalWritable := 'False'} : Bool;   // Detection is not off
      AlarmCondReqOn { ExternalAccessible := 'False'; ExternalVisible := 'False'; ExternalWritable := 'False'} : Bool;   // Alarm condition
      AlarmCondReqOff { ExternalAccessible := 'False'; ExternalVisible := 'False'; ExternalWritable := 'False'} : Bool;   // Alarm condition
   END_VAR
BEGIN

REGION Network 1: **** 2.2 - Alarms - Alarm generation **** Condition alarm for active signal
   // Condition alarm for active signal
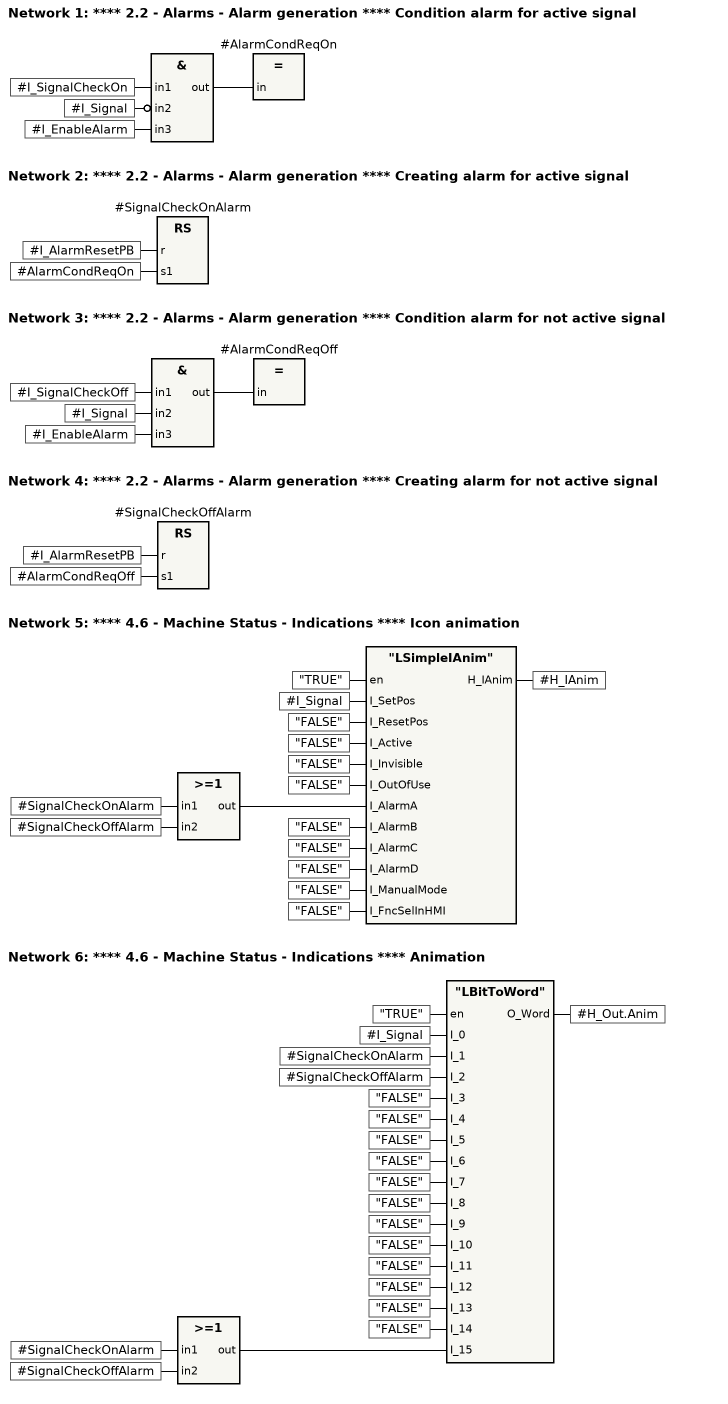
   #AlarmCondReqOn := #I_SignalCheckOn AND NOT #I_Signal AND #I_EnableAlarm;
END_REGION

REGION Network 2: **** 2.2 - Alarms - Alarm generation **** Creating alarm for active signal
   // Creating alarm for active signal
   IF #I_AlarmResetPB THEN
       #SignalCheckOnAlarm := FALSE;   // RS flip-flop
   END_IF;
   IF #AlarmCondReqOn THEN #SignalCheckOnAlarm := TRUE; END_IF;
END_REGION

REGION Network 3: **** 2.2 - Alarms - Alarm generation **** Condition alarm for not active signal
   // Condition alarm for not active signal
   #AlarmCondReqOff := #I_SignalCheckOff AND #I_Signal AND #I_EnableAlarm;
END_REGION

REGION Network 4: **** 2.2 - Alarms - Alarm generation **** Creating alarm for not active signal
   // Creating alarm for not active signal
   IF #I_AlarmResetPB THEN
       #SignalCheckOffAlarm := FALSE;   // RS flip-flop
   END_IF;
   IF #AlarmCondReqOff THEN #SignalCheckOffAlarm := TRUE; END_IF;
END_REGION

REGION Network 5: **** 4.6 - Machine Status - Indications **** Icon animation
   // Icon animation
   IF "TRUE" THEN
       "LSimpleIAnim"(I_SetPos := #I_Signal,
                      I_ResetPos := "FALSE",
                      I_Active := "FALSE",
                      I_Invisible := "FALSE",
                      I_OutOfUse := "FALSE",
                      I_AlarmA := #SignalCheckOnAlarm OR #SignalCheckOffAlarm,
                      I_AlarmB := "FALSE",
                      I_AlarmC := "FALSE",
                      I_AlarmD := "FALSE",
                      I_ManualMode := "FALSE",
                      I_FncSelInHMI := "FALSE",
                      H_IAnim => #H_IAnim);
   END_IF;
END_REGION

REGION Network 6: **** 4.6 - Machine Status - Indications **** Animation
   // Animation
   IF "TRUE" THEN
       "LBitToWord"(I_0 := #I_Signal,
                    I_1 := #SignalCheckOnAlarm,
                    I_2 := #SignalCheckOffAlarm,
                    I_3 := "FALSE",
                    I_4 := "FALSE",
                    I_5 := "FALSE",
                    I_6 := "FALSE",
                    I_7 := "FALSE",
                    I_8 := "FALSE",
                    I_9 := "FALSE",
                    I_10 := "FALSE",
                    I_11 := "FALSE",
                    I_12 := "FALSE",
                    I_13 := "FALSE",
                    I_14 := "FALSE",
                    I_15 := #SignalCheckOnAlarm OR #SignalCheckOffAlarm,
                    O_Word => #H_Out.Anim);
   END_IF;
END_REGION

REGION Network 7: *** 8 - Outputs ***** Signal on
   // Signal on
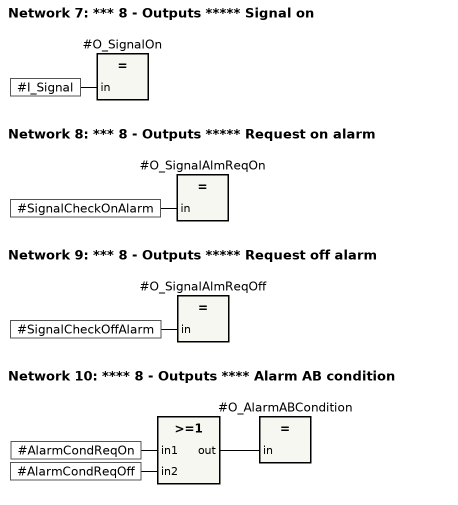
   #O_SignalOn := #I_Signal;
END_REGION

REGION Network 8: *** 8 - Outputs ***** Request on alarm
   // Request on alarm
   #O_SignalAlmReqOn := #SignalCheckOnAlarm;
END_REGION

REGION Network 9: *** 8 - Outputs ***** Request off alarm
   // Request off alarm
   #O_SignalAlmReqOff := #SignalCheckOffAlarm;
END_REGION

REGION Network 10: **** 8 - Outputs **** Alarm AB condition
   // Alarm AB condition
   #O_AlarmABCondition := #AlarmCondReqOn OR #AlarmCondReqOff;
END_REGION
END_FUNCTION_BLOCK

FUNCTION_BLOCK "LVIDSMaster"   // FB1201, SCL
TITLE = LVIDSMaster
{ S7_Optimized_Access := 'FALSE' }
VERSION : 0.1
// stored: AutoNumber false, IsIECCheckEnabled false, SetENOAutomatically False, UDAEnableTagReadback false
   VAR_INPUT
      C_SubSystem { ExternalAccessible := 'False'; ExternalVisible := 'False'; ExternalWritable := 'False'} : Int;   // VDComm - Subsystem
      C_VDCommMasterRcvDB { ExternalAccessible := 'False'; ExternalVisible := 'False'; ExternalWritable := 'False'} : DB_ANY;   // VDComm - Master receive DB
      C_VDCommMasterSndDB { ExternalAccessible := 'False'; ExternalVisible := 'False'; ExternalWritable := 'False'} : DB_ANY;   // VDComm - Master send DB
      C_VDCommLocalRcvDB { ExternalAccessible := 'False'; ExternalVisible := 'False'; ExternalWritable := 'False'} : DB_ANY;   // VDComm - Local receive DB
      C_VDCommLocalSndDB { ExternalAccessible := 'False'; ExternalVisible := 'False'; ExternalWritable := 'False'} : DB_ANY;   // VDComm - Local send DB
      C_Plant { ExternalAccessible := 'False'; ExternalVisible := 'False'; ExternalWritable := 'False'} : Int;   // Plant ( VCG : 321, VCT : 461, VCCD : 861, VCQD : 862, VCLQ : 863, VCCH : 11 )
      C_IDType { ExternalAccessible := 'False'; ExternalVisible := 'False'; ExternalWritable := 'False'} : DWord;   // Identifier type (0 : Body tag, > 0 : Carrier tag Ex.: Carrier A-shop 162)
      I_OutOfUse { ExternalAccessible := 'False'; ExternalVisible := 'False'; ExternalWritable := 'False'} : Bool;   // Put out of use
      I_PartPres { ExternalAccessible := 'False'; ExternalVisible := 'False'; ExternalWritable := 'False'} : Bool;   // Cycle of tag data use active / Part is present in station
      I_TagID { ExternalAccessible := 'False'; ExternalVisible := 'False'; ExternalWritable := 'False'} : DWord;   // Tag identification ( to get VEM data )
      I_BodyID { ExternalAccessible := 'False'; ExternalVisible := 'False'; ExternalWritable := 'False'} : DWord;   // Body identification ( to get VEM data )
      I_CarrierID { ExternalAccessible := 'False'; ExternalVisible := 'False'; ExternalWritable := 'False'} : DWord;   // Carrier identification ( to get VEM data )
      I_MixNbr { ExternalAccessible := 'False'; ExternalVisible := 'False'; ExternalWritable := 'False'} : DWord;   // Mixnumber ( to get VEM data )
      I_PopID { ExternalAccessible := 'False'; ExternalVisible := 'False'; ExternalWritable := 'False'} : UDInt;   // Spare Data / PopID ( to get VEM data )
      I_PopIDSuffix { ExternalAccessible := 'False'; ExternalVisible := 'False'; ExternalWritable := 'False'} : Char;   // PopID suffix ( to get VEM data )
      I_PopType { ExternalAccessible := 'False'; ExternalVisible := 'False'; ExternalWritable := 'False'} : UDInt;   // Pop identifier ( to get VEM data )
      I_StartGetVEMData { ExternalAccessible := 'False'; ExternalVisible := 'False'; ExternalWritable := 'False'} : Bool;   // Get VEM data - Start on edge
      I_ResetAlarm { ExternalAccessible := 'False'; ExternalVisible := 'False'; ExternalWritable := 'False'} : Bool;   // Reset alarm
   END_VAR
   VAR_OUTPUT
      O_VEMDataValid { ExternalAccessible := 'False'; ExternalVisible := 'False'; ExternalWritable := 'False'} : Bool;   // VEM data is valid
      O_VEMDataNotValid { ExternalAccessible := 'False'; ExternalVisible := 'False'; ExternalWritable := 'False'} : Bool;   // VEM data is not valid
      O_GetVEMDataBusy { ExternalAccessible := 'False'; ExternalVisible := 'False'; ExternalWritable := 'False'} : Bool;   // Get VEM data - Busy
      O_Status { ExternalAccessible := 'False'; ExternalVisible := 'False'; ExternalWritable := 'False'} : Int;   // 0: no activity, 1: OK-Data valid, 2: Busy, -1..-32768: error code / 0: no activity, 1: OK-Get VEM data valid, 2: Busy, -1..-32768: error code
      O_Alarm { ExternalAccessible := 'False'; ExternalVisible := 'False'; ExternalWritable := 'False'} : Bool;   // Get VEM Data Alarm (Status < 0)
   END_VAR
   VAR_IN_OUT
      IO_VDComm : "VDComm";   // VD Comm / VD Comm - communication record
      IO_VIDS : "VIDS";   // VIDS - internal record
      IO_VEMData : "VEMData";   // VEM data - received
      IO_VEMDataChange : "VEMData";   // VEM data - to be changed
      IO_SpecificData : Array[0..7925] of Byte;   // Specific data received
      IO_Alarm : "Alarm";   // Alarm
      H_Master : "H_LVIDSMaster";   // Animation
      H_HMI : "H_HMI";   // Used for icon animation
   END_VAR
   VAR DB_SPECIFIC
      i { ExternalAccessible := 'False'; ExternalVisible := 'False'; ExternalWritable := 'False'} : Int;   // Index
      PartPres { ExternalAccessible := 'False'; ExternalVisible := 'False'; ExternalWritable := 'False'} : Bool;
      PartLostDlyTmrElapsed { ExternalAccessible := 'False'; ExternalVisible := 'False'; ExternalWritable := 'False'} : Bool;
      PartLostDlyTmrAct { ExternalAccessible := 'False'; ExternalVisible := 'False'; ExternalWritable := 'False'} : DInt;
      VEMDataChangeIoSerial { ExternalAccessible := 'False'; ExternalVisible := 'False'; ExternalWritable := 'False'} : Bool;
      VEMDataChangeHMISerial { ExternalAccessible := 'False'; ExternalVisible := 'False'; ExternalWritable := 'False'} : Array[0..255] of Byte;
      VEMDataChangeHMI { ExternalAccessible := 'False'; ExternalVisible := 'False'; ExternalWritable := 'False'; S7_SetPoint := 'True'} : "VEMData";
      VEMDataInitArray { ExternalAccessible := 'False'; ExternalVisible := 'False'; ExternalWritable := 'False'} : Array[0..255] of Byte;   // VEM data in serialized form
      VEMDataRcvArray { ExternalAccessible := 'False'; ExternalVisible := 'False'; ExternalWritable := 'False'} : Array[0..255] of Byte;   // VEM data in serialized form
      VEMDataRcv { ExternalAccessible := 'False'; ExternalVisible := 'False'; ExternalWritable := 'False'; S7_SetPoint := 'True'} : "VEMData";
      VEMDataSndArray { ExternalAccessible := 'False'; ExternalVisible := 'False'; ExternalWritable := 'False'} : Array[0..255] of Byte;
      SpecificData { ExternalAccessible := 'False'; ExternalVisible := 'False'; ExternalWritable := 'False'} : Array[0..7925] of Byte;
      VEMDataValid { ExternalAccessible := 'False'; ExternalVisible := 'False'; ExternalWritable := 'False'} : Bool;
      VEMDataNotValid { ExternalAccessible := 'False'; ExternalVisible := 'False'; ExternalWritable := 'False'} : Bool;
      CmdCodeSent { ExternalAccessible := 'False'; ExternalVisible := 'False'; ExternalWritable := 'False'} : DWord;   // Command code sent to VD
      CmdCodeRcvd { ExternalAccessible := 'False'; ExternalVisible := 'False'; ExternalWritable := 'False'} : DWord;   // Command code received from VD
      TagIDMem { ExternalAccessible := 'False'; ExternalVisible := 'False'; ExternalWritable := 'False'} : DWord;
      BodyIDMem { ExternalAccessible := 'False'; ExternalVisible := 'False'; ExternalWritable := 'False'} : DWord;
      CarrierIDMem { ExternalAccessible := 'False'; ExternalVisible := 'False'; ExternalWritable := 'False'} : DWord;
      MixNbrMem { ExternalAccessible := 'False'; ExternalVisible := 'False'; ExternalWritable := 'False'} : DWord;
      PopIDMem { ExternalAccessible := 'False'; ExternalVisible := 'False'; ExternalWritable := 'False'} : UDInt;   // Spare Data / PopID
      PopIDSuffixMem { ExternalAccessible := 'False'; ExternalVisible := 'False'; ExternalWritable := 'False'} : Char;   // PopID suffix
      PopTypeMem { ExternalAccessible := 'False'; ExternalVisible := 'False'; ExternalWritable := 'False'} : UDInt;   // Spare Data / Pop Identifier
      CarTypeVariant { ExternalAccessible := 'False'; ExternalVisible := 'False'; ExternalWritable := 'False'} : Int;   // Car type - Decoded from variant
      CarTypeBody { ExternalAccessible := 'False'; ExternalVisible := 'False'; ExternalWritable := 'False'} : Int;   // Car type - Decoded from bodytype matrix
      SteeringVariant { ExternalAccessible := 'False'; ExternalVisible := 'False'; ExternalWritable := 'False'} : Int;
      SteeringBody { ExternalAccessible := 'False'; ExternalVisible := 'False'; ExternalWritable := 'False'} : Int;
      CarTypeArray { ExternalAccessible := 'False'; ExternalVisible := 'False'; ExternalWritable := 'False'} : Array[1..3] of Int;
      DataValidSnd { ExternalAccessible := 'False'; ExternalVisible := 'False'; ExternalWritable := 'False'} : Bool;   // Data valid - Send
      DataRcvOk { ExternalAccessible := 'False'; ExternalVisible := 'False'; ExternalWritable := 'False'} : Bool;
      DataRcvNok { ExternalAccessible := 'False'; ExternalVisible := 'False'; ExternalWritable := 'False'} : Bool;
      DeserializePos { ExternalAccessible := 'False'; ExternalVisible := 'False'; ExternalWritable := 'False'} : DInt;
      SerializePos { ExternalAccessible := 'False'; ExternalVisible := 'False'; ExternalWritable := 'False'} : DInt;
      SequenceTotalOvertime { ExternalAccessible := 'False'; ExternalVisible := 'False'; ExternalWritable := 'False'} : Time;
      StartChangeVEMDataEdg { ExternalAccessible := 'False'; ExternalVisible := 'False'; ExternalWritable := 'False'} : Bool;   // Change VEM data - Start edge
      StartChangeVEMDataPls { ExternalAccessible := 'False'; ExternalVisible := 'False'; ExternalWritable := 'False'} : Bool;   // Change VEM data - Start pulse
      SeqOvTimeElapsed { ExternalAccessible := 'False'; ExternalVisible := 'False'; ExternalWritable := 'False'} : Bool;
      CodeBusy { ExternalAccessible := 'False'; ExternalVisible := 'False'; ExternalWritable := 'False'} : Int;
      RetVal { ExternalAccessible := 'False'; ExternalVisible := 'False'; ExternalWritable := 'False'} : Int;   // Return value
      GetVEMDataByRFIDBeginReqEdg { ExternalAccessible := 'False'; ExternalVisible := 'False'; ExternalWritable := 'False'} : Bool;
      GetVEMDataByTagReplBeginReqEdg { ExternalAccessible := 'False'; ExternalVisible := 'False'; ExternalWritable := 'False'} : Bool;
      DataValidRcvGetVEMDataByRFID { ExternalAccessible := 'False'; ExternalVisible := 'False'; ExternalWritable := 'False'} : Bool;
      GetVEMDataBeginReqEdg { ExternalAccessible := 'False'; ExternalVisible := 'False'; ExternalWritable := 'False'} : Bool;
      GetVEMDataByHMIBeginEdg { ExternalAccessible := 'False'; ExternalVisible := 'False'; ExternalWritable := 'False'} : Bool;
      GetVEMDataRcvOk { ExternalAccessible := 'False'; ExternalVisible := 'False'; ExternalWritable := 'False'} : Bool;
      ChangeDataReq { ExternalAccessible := 'False'; ExternalVisible := 'False'; ExternalWritable := 'False'} : Bool;
      ChangeDataReqEdg { ExternalAccessible := 'False'; ExternalVisible := 'False'; ExternalWritable := 'False'} : Bool;
      ChangeDataBeginReqEdg { ExternalAccessible := 'False'; ExternalVisible := 'False'; ExternalWritable := 'False'} : Bool;
      ChangeDataRcvOk { ExternalAccessible := 'False'; ExternalVisible := 'False'; ExternalWritable := 'False'} : Bool;
      GetNextIDBeginReqEdg { ExternalAccessible := 'False'; ExternalVisible := 'False'; ExternalWritable := 'False'} : Bool;
      GetNextIDRcvOk { ExternalAccessible := 'False'; ExternalVisible := 'False'; ExternalWritable := 'False'} : Bool;
      ReplaceTagReq { ExternalAccessible := 'False'; ExternalVisible := 'False'; ExternalWritable := 'False'} : Bool;
      ReplaceTagReqEdg { ExternalAccessible := 'False'; ExternalVisible := 'False'; ExternalWritable := 'False'} : Bool;
      ReplaceTagBeginReqEdg { ExternalAccessible := 'False'; ExternalVisible := 'False'; ExternalWritable := 'False'} : Bool;
      ReplaceTagRcvOk { ExternalAccessible := 'False'; ExternalVisible := 'False'; ExternalWritable := 'False'} : Bool;
      InitTagBeginReqEdg { ExternalAccessible := 'False'; ExternalVisible := 'False'; ExternalWritable := 'False'} : Bool;
      InitTagRcvOk { ExternalAccessible := 'False'; ExternalVisible := 'False'; ExternalWritable := 'False'} : Bool;
      GetSpecDataReq { ExternalAccessible := 'False'; ExternalVisible := 'False'; ExternalWritable := 'False'} : Bool;
      GetSpecDataReqEdg { ExternalAccessible := 'False'; ExternalVisible := 'False'; ExternalWritable := 'False'} : Bool;
      GetSpecDataBeginReqEdg { ExternalAccessible := 'False'; ExternalVisible := 'False'; ExternalWritable := 'False'} : Bool;
      GetSpecDataRcvOk { ExternalAccessible := 'False'; ExternalVisible := 'False'; ExternalWritable := 'False'} : Bool;
      PutSpecDataBeginReqEdg { ExternalAccessible := 'False'; ExternalVisible := 'False'; ExternalWritable := 'False'} : Bool;
      PutSpecDataRcvOk { ExternalAccessible := 'False'; ExternalVisible := 'False'; ExternalWritable := 'False'} : Bool;
      TrackBeginReqEdg { ExternalAccessible := 'False'; ExternalVisible := 'False'; ExternalWritable := 'False'} : Bool;   // Tracking - Begin request edge
      TrackingRcvOk { ExternalAccessible := 'False'; ExternalVisible := 'False'; ExternalWritable := 'False'} : Bool;
      CoupleBeginReqEdg { ExternalAccessible := 'False'; ExternalVisible := 'False'; ExternalWritable := 'False'} : Bool;
      CoupleRcvOk { ExternalAccessible := 'False'; ExternalVisible := 'False'; ExternalWritable := 'False'} : Bool;
      DecoupleBeginReqEdg { ExternalAccessible := 'False'; ExternalVisible := 'False'; ExternalWritable := 'False'} : Bool;
      DecoupleRcvOk { ExternalAccessible := 'False'; ExternalVisible := 'False'; ExternalWritable := 'False'} : Bool;
      ConfirmBeginReqEdg { ExternalAccessible := 'False'; ExternalVisible := 'False'; ExternalWritable := 'False'} : Bool;
      ConfirmationRcvOk { ExternalAccessible := 'False'; ExternalVisible := 'False'; ExternalWritable := 'False'} : Bool;
      NoFunctionBusy { ExternalAccessible := 'False'; ExternalVisible := 'False'; ExternalWritable := 'False'} : Bool;
      Busy { ExternalAccessible := 'False'; ExternalVisible := 'False'; ExternalWritable := 'False'} : Bool;
      BtnGetVEMTagIDEdge { ExternalAccessible := 'False'; ExternalVisible := 'False'; ExternalWritable := 'False'} : Bool;
      btnGetVEMDataByMixNbrEdg { ExternalAccessible := 'False'; ExternalVisible := 'False'; ExternalWritable := 'False'} : Bool;
      BtnGetVEMCarrierEdge { ExternalAccessible := 'False'; ExternalVisible := 'False'; ExternalWritable := 'False'} : Bool;
      ChangeDataNotValid { ExternalAccessible := 'False'; ExternalVisible := 'False'; ExternalWritable := 'False'} : Bool;
      MessageLength { ExternalAccessible := 'False'; ExternalVisible := 'False'; ExternalWritable := 'False'} : Word;   // Message Length
      SendToVD { ExternalAccessible := 'False'; ExternalVisible := 'False'; ExternalWritable := 'False'} : Bool;   // Send To PCS
      SendFinished { ExternalAccessible := 'False'; ExternalVisible := 'False'; ExternalWritable := 'False'} : Bool;   // Send Finished / Send data Finished
      RcvOkGetVEMDataCode { ExternalAccessible := 'False'; ExternalVisible := 'False'; ExternalWritable := 'False'} : Bool;
      RcvOkIdentification { ExternalAccessible := 'False'; ExternalVisible := 'False'; ExternalWritable := 'False'} : Bool;
      NewData { ExternalAccessible := 'False'; ExternalVisible := 'False'; ExternalWritable := 'False'} : Bool;   // New Data Is Present
      ResetNewData { ExternalAccessible := 'False'; ExternalVisible := 'False'; ExternalWritable := 'False'} : Bool;   // Reset Data Recevied
      CarrierIDDataReqOk { ExternalAccessible := 'False'; ExternalVisible := 'False'; ExternalWritable := 'False'} : Bool;
      ReqSendReport { ExternalAccessible := 'False'; ExternalVisible := 'False'; ExternalWritable := 'False'} : Bool;
      SendCmd { ExternalAccessible := 'False'; ExternalVisible := 'False'; ExternalWritable := 'False'} : Bool;   // External command send
      ResetAllRequests { ExternalAccessible := 'False'; ExternalVisible := 'False'; ExternalWritable := 'False'} : Bool;
      HMIGetVEMDataTagIDMem { ExternalAccessible := 'False'; ExternalVisible := 'False'; ExternalWritable := 'False'} : DInt;
      HMIGetVEMDataMixNbrMem { ExternalAccessible := 'False'; ExternalVisible := 'False'; ExternalWritable := 'False'} : DInt;
      HMIGetVEMDataCarrIdMem { ExternalAccessible := 'False'; ExternalVisible := 'False'; ExternalWritable := 'False'} : DInt;
      StartGetVEMDataEdg { ExternalAccessible := 'False'; ExternalVisible := 'False'; ExternalWritable := 'False'} : Bool;
      StartGetVEMDataPls { ExternalAccessible := 'False'; ExternalVisible := 'False'; ExternalWritable := 'False'} : Bool;
      Status { ExternalAccessible := 'False'; ExternalVisible := 'False'; ExternalWritable := 'False'} : Int;
      StatusMem { ExternalAccessible := 'False'; ExternalVisible := 'False'; ExternalWritable := 'False'} : Int;
      StepNbr { ExternalAccessible := 'False'; ExternalVisible := 'False'; ExternalWritable := 'False'} : Int;   // Active stepnumber
      Step0ExitPls { ExternalAccessible := 'False'; ExternalVisible := 'False'; ExternalWritable := 'False'} : Bool;   // Step 0 - Pulse created on exit
      Step50EntryEdg { ExternalAccessible := 'False'; ExternalVisible := 'False'; ExternalWritable := 'False'} : Bool;   // Step 50 - Edge created on entry
      Step50EntryPls { ExternalAccessible := 'False'; ExternalVisible := 'False'; ExternalWritable := 'False'} : Bool;   // Step 50 - Pulse created on entry
      Step50ExitEdg { ExternalAccessible := 'False'; ExternalVisible := 'False'; ExternalWritable := 'False'} : Bool;   // Step 50 - Edge created on exit
      Step50ExitPls { ExternalAccessible := 'False'; ExternalVisible := 'False'; ExternalWritable := 'False'} : Bool;   // Step 50 - Pulse created on exit
      Step100EntryEdg { ExternalAccessible := 'False'; ExternalVisible := 'False'; ExternalWritable := 'False'} : Bool;   // Step 100 - Edge created on entry
      Step100EntryPls { ExternalAccessible := 'False'; ExternalVisible := 'False'; ExternalWritable := 'False'} : Bool;   // Step 100 - Pulse created on entry
      Step100ExitEdg { ExternalAccessible := 'False'; ExternalVisible := 'False'; ExternalWritable := 'False'} : Bool;   // Step 100 - Edge created on exit
      Step100ExitPls { ExternalAccessible := 'False'; ExternalVisible := 'False'; ExternalWritable := 'False'} : Bool;   // Step 100 - Pulse created on exit
      Step200EntryEdg { ExternalAccessible := 'False'; ExternalVisible := 'False'; ExternalWritable := 'False'} : Bool;   // Step 200 - Edge created on entry
      Step200EntryPls { ExternalAccessible := 'False'; ExternalVisible := 'False'; ExternalWritable := 'False'} : Bool;   // Step 200 - Pulse created on entry
      Step200ExitEdg { ExternalAccessible := 'False'; ExternalVisible := 'False'; ExternalWritable := 'False'} : Bool;   // Step 200 - Edge created on exit
      Step200ExitPls { ExternalAccessible := 'False'; ExternalVisible := 'False'; ExternalWritable := 'False'} : Bool;   // Step 200 - Pulse created on exit
      Step300EntryEdg { ExternalAccessible := 'False'; ExternalVisible := 'False'; ExternalWritable := 'False'} : Bool;   // Step 300 - Edge created on entry
      Step300EntryPls { ExternalAccessible := 'False'; ExternalVisible := 'False'; ExternalWritable := 'False'} : Bool;   // Step 300 - Pulse created on entry
      Step300ExitEdg { ExternalAccessible := 'False'; ExternalVisible := 'False'; ExternalWritable := 'False'} : Bool;   // Step 300 - Edge created on exit
      Step300ExitPls { ExternalAccessible := 'False'; ExternalVisible := 'False'; ExternalWritable := 'False'} : Bool;   // Step 300 - Pulse created on exit
      Step400ExitEdg { ExternalAccessible := 'False'; ExternalVisible := 'False'; ExternalWritable := 'False'} : Bool;   // Step 400 - Edge created on exit
      Step400ExitPls { ExternalAccessible := 'False'; ExternalVisible := 'False'; ExternalWritable := 'False'} : Bool;   // Step 400 - Pulse created on exit
      Step0To50Cond { ExternalAccessible := 'False'; ExternalVisible := 'False'; ExternalWritable := 'False'} : Bool;   // Step 0 to 50 - Condition
      Step50To100Cond { ExternalAccessible := 'False'; ExternalVisible := 'False'; ExternalWritable := 'False'} : Bool;   // Step 0 to 100 - Condition
      Step50To200Cond { ExternalAccessible := 'False'; ExternalVisible := 'False'; ExternalWritable := 'False'} : Bool;   // Step 0 to 200 - Condition
      Step100To300Cond1 { ExternalAccessible := 'False'; ExternalVisible := 'False'; ExternalWritable := 'False'} : Bool;   // Step 100 to 300 - Condition 1
      Step100To300Cond2 { ExternalAccessible := 'False'; ExternalVisible := 'False'; ExternalWritable := 'False'} : Bool;   // Step 100 to 300 - Condition 2
      Step100To300Cond { ExternalAccessible := 'False'; ExternalVisible := 'False'; ExternalWritable := 'False'} : Bool;   // Step 100 to 300 - Condition
      Step200To300Cond { ExternalAccessible := 'False'; ExternalVisible := 'False'; ExternalWritable := 'False'} : Bool;   // Step 200 to 300 - Condition
      Step300To400Cond { ExternalAccessible := 'False'; ExternalVisible := 'False'; ExternalWritable := 'False'} : Bool;   // Step 300 to 400 - Condition
      Step300To400Cond1 { ExternalAccessible := 'False'; ExternalVisible := 'False'; ExternalWritable := 'False'} : Bool;   // Step 300 to 400 - Condition 1
      Step300To400Cond2 { ExternalAccessible := 'False'; ExternalVisible := 'False'; ExternalWritable := 'False'} : Bool;   // Step 300 to 400 - Condition 2
      Step400To0Cond { ExternalAccessible := 'False'; ExternalVisible := 'False'; ExternalWritable := 'False'} : Bool;   // Step 400 to 0 - Condition
      DataRcvOkGetSpecData { ExternalAccessible := 'False'; ExternalVisible := 'False'; ExternalWritable := 'False'} : Bool;
      VEMDataRcvOKCond1 { ExternalAccessible := 'False'; ExternalVisible := 'False'; ExternalWritable := 'False'} : Bool;
      VEMDataRcvOKCond2 { ExternalAccessible := 'False'; ExternalVisible := 'False'; ExternalWritable := 'False'} : Bool;
      VDCommLocalSndDB { ExternalAccessible := 'False'; ExternalVisible := 'False'; ExternalWritable := 'False'} : Int;   // Send DB / VD Comm - Local send DB number
      VDCommLocalRcvDB { ExternalAccessible := 'False'; ExternalVisible := 'False'; ExternalWritable := 'False'} : Int;   // Recv DB / VD Comm - Local receive DB number
      VD_Identification { ExternalAccessible := 'False'; ExternalVisible := 'False'; ExternalWritable := 'False'} : DWord;   // Identification from VD
      SpecDataLength_DW { ExternalAccessible := 'False'; ExternalVisible := 'False'; ExternalWritable := 'False'} : DWord;
      SpecDataLength_DInt { ExternalAccessible := 'False'; ExternalVisible := 'False'; ExternalWritable := 'False'} : DInt;
      TotalDataSentLength { ExternalAccessible := 'False'; ExternalVisible := 'False'; ExternalWritable := 'False'} : DInt;
      Cmd { ExternalAccessible := 'False'; ExternalVisible := 'False'; ExternalWritable := 'False'} : DWord;
      SeqOvTime { ExternalAccessible := 'False'; ExternalVisible := 'False'; ExternalWritable := 'False'} : Bool;
      OkBegin { ExternalAccessible := 'False'; ExternalVisible := 'False'; ExternalWritable := 'False'} : Bool;
      Step50TmrElapsed { ExternalAccessible := 'False'; ExternalVisible := 'False'; ExternalWritable := 'False'} : Bool;   // Step 50 - Step time elapsed
      Step50TmrAct { ExternalAccessible := 'False'; ExternalVisible := 'False'; ExternalWritable := 'False'} : DInt;   // Step 50 - Step time actual
      Step50TmrActMax { ExternalAccessible := 'False'; ExternalVisible := 'False'; ExternalWritable := 'False'} : DInt;   // Step 50 - Step time actual maximum
      Step100TmrElapsed { ExternalAccessible := 'False'; ExternalVisible := 'False'; ExternalWritable := 'False'} : Bool;   // Step 100 - Step time elapsed
      Step100TmrAct { ExternalAccessible := 'False'; ExternalVisible := 'False'; ExternalWritable := 'False'} : DInt;   // Step 100 - Step time actual
      Step100TmrActMax { ExternalAccessible := 'False'; ExternalVisible := 'False'; ExternalWritable := 'False'} : DInt;   // Step 100 - Step time actual maximum
      Step200TmrElapsed { ExternalAccessible := 'False'; ExternalVisible := 'False'; ExternalWritable := 'False'} : Bool;   // Step 200 - Step time elapsed
      Step200TmrAct { ExternalAccessible := 'False'; ExternalVisible := 'False'; ExternalWritable := 'False'} : DInt;   // Step 200 - Step time actual
      Step200TmrActMax { ExternalAccessible := 'False'; ExternalVisible := 'False'; ExternalWritable := 'False'} : DInt;   // Step 200 - Step time actual maximum
      Step300TmrElapsed { ExternalAccessible := 'False'; ExternalVisible := 'False'; ExternalWritable := 'False'} : Bool;   // Step 300 - Step time elapsed
      Step300TmrAct { ExternalAccessible := 'False'; ExternalVisible := 'False'; ExternalWritable := 'False'} : DInt;   // Step 300 - Step time actual
      Step300TmrActMax { ExternalAccessible := 'False'; ExternalVisible := 'False'; ExternalWritable := 'False'} : DInt;   // Step 300 - Step time actual maximum
      Step400TmrElapsed { ExternalAccessible := 'False'; ExternalVisible := 'False'; ExternalWritable := 'False'} : Bool;   // Step 400 - Step time elapsed
      Step400TmrAct { ExternalAccessible := 'False'; ExternalVisible := 'False'; ExternalWritable := 'False'} : DInt;   // Step 400 - Step time actual
      Step400TmrActMax { ExternalAccessible := 'False'; ExternalVisible := 'False'; ExternalWritable := 'False'} : DInt;   // Step 400 - Step time actual maximum
      EmptyByte { ExternalAccessible := 'False'; ExternalVisible := 'False'; ExternalWritable := 'False'} : Byte;
      PartLostEdg { ExternalAccessible := 'False'; ExternalVisible := 'False'; ExternalWritable := 'False'} : Bool;   // Part lost edge
      PartLostPls { ExternalAccessible := 'False'; ExternalVisible := 'False'; ExternalWritable := 'False'} : Bool;   // Part lost pulse
      PutVemDataTotalLength { ExternalAccessible := 'False'; ExternalVisible := 'False'; ExternalWritable := 'False'} : DInt;
      DataValidRcv { ExternalAccessible := 'False'; ExternalVisible := 'False'; ExternalWritable := 'False'} : Bool;
      BusyGetVEMData { ExternalAccessible := 'False'; ExternalVisible := 'False'; ExternalWritable := 'False'} : Bool;
      Alarm { ExternalAccessible := 'False'; ExternalVisible := 'False'; ExternalWritable := 'False'} : Bool;   // Alarm
      msgPartPresVisible { ExternalAccessible := 'False'; ExternalVisible := 'False'; ExternalWritable := 'False'} : Word;   // HMI - Message animation - Part present - Visible
      msgPartPresAnim { ExternalAccessible := 'False'; ExternalVisible := 'False'; ExternalWritable := 'False'} : Word;   // HMI - Message animation - Part present - Summary
      msgPartNotPresVisible { ExternalAccessible := 'False'; ExternalVisible := 'False'; ExternalWritable := 'False'} : Word;   // HMI - Message animation - Part not present - Visible
      msgPartNotPresAnim { ExternalAccessible := 'False'; ExternalVisible := 'False'; ExternalWritable := 'False'} : Word;   // HMI - Message animation - Part not present - Summary
      IconColour { ExternalAccessible := 'False'; ExternalVisible := 'False'; ExternalWritable := 'False'} : Word;   // Icon colour
      SPACE { ExternalAccessible := 'False'; ExternalVisible := 'False'; ExternalWritable := 'False'} : Char := ' ';
   END_VAR
   VAR
      _Step50Tmr { ExternalAccessible := 'False'; ExternalVisible := 'False'; ExternalWritable := 'False'; S7_SetPoint := 'True'} : "LTimer";   // Step 50 - Timer
      _Step100Tmr { ExternalAccessible := 'False'; ExternalVisible := 'False'; ExternalWritable := 'False'; S7_SetPoint := 'True'} : "LTimer";   // Step 100 - Timer
      _Step200Tmr { ExternalAccessible := 'False'; ExternalVisible := 'False'; ExternalWritable := 'False'; S7_SetPoint := 'True'} : "LTimer";   // Step 200 - Timer
      _Step300Tmr { ExternalAccessible := 'False'; ExternalVisible := 'False'; ExternalWritable := 'False'; S7_SetPoint := 'True'} : "LTimer";   // Step 300 - Timer
      "_LVDComSubSystemS7-1500" { ExternalAccessible := 'False'; ExternalVisible := 'False'; ExternalWritable := 'False'; S7_SetPoint := 'True'} : "LVDComSubSystemS7-1500";
      _PartLostDlyTmr { ExternalAccessible := 'False'; ExternalVisible := 'False'; ExternalWritable := 'False'; S7_SetPoint := 'True'} : "LTimer";   // Part present lost delay timer
   END_VAR
   VAR_TEMP
      ptrIO_VEMData : Any;   // Pointer to received VEM data / Pointer to IO_VEM data
      ptrIO_VEMDataStruct AT ptrIO_VEMData : Struct   // Pointer to IO_VEM data - Structure
         ID : Byte;
         DataType : Byte;
         ReplicationFactor : Word;
         DbNbr : Word;
         CrossAreaPointer : DWord;
      END_STRUCT;
      ptrIO_VEMDataChange : Any;   // Pointer to received VEM data / Pointer to IO_VEM data Change
      ptrIO_VEMDataChangeStruct AT ptrIO_VEMDataChange : Struct   // Pointer to IO_VEM data Change - Structure
         ID : Byte;
         DataType : Byte;
         ReplicationFactor : Word;
         DbNbr : Word;
         CrossAreaPointer : DWord;
      END_STRUCT;
      ptrIO_SpecData : Any;   // Pointer to received VEM data / Pointer to IO_Specific data
      ptrIO_SpecDataStruct AT ptrIO_SpecData : Struct   // Pointer to IO_Specific data - Structure
         ID : Byte;
         DataType : Byte;
         ReplicationFactor : Word;
         DbNbr : Word;
         CrossAreaPointer : DWord;
      END_STRUCT;
      ptrVEMDataVDCommLocalRcv : Any;   // Pointer to received VEM data / Pointer to VEM data in VD local receive DB
      ptrVEMDataVDCommLocalRcvStruct AT ptrVEMDataVDCommLocalRcv : Struct   // Pointer to VEM data in VD local receive DB - Structure
         ID : Byte;
         DataType : Byte;
         ReplicationFactor : Word;
         DbNbr : Word;
         CrossAreaPointer : DWord;
      END_STRUCT;
      ptrVEMDataVDCommLocalSnd : Any;   // Pointer to VEM and specific data to be sent / Pointer to VEM data in VD local send DB
      ptrVEMDataVDCommLocalSndStruct AT ptrVEMDataVDCommLocalSnd : Struct   // Pointer to VEM data in VD local send DB - Structure
         ID : Byte;
         DataType : Byte;
         ReplicationFactor : Word;
         DbNbr : Word;
         CrossAreaPointer : DWord;
      END_STRUCT;
      ptrSpecDataVDCommLocalRcv : Any;   // Pointer to received specific data / Pointer to Specific data in VD local receive DB
      ptrSpecDataVDCommLocalRcvStruct AT ptrSpecDataVDCommLocalRcv : Struct   // Pointer to Specific data in VD local receive DB - Structure
         ID : Byte;
         DataType : Byte;
         ReplicationFactor : Word;
         DbNbr : Word;
         CrossAreaPointer : DWord;
      END_STRUCT;
      ptrSpecDataVDCommLocalSnd : Any;   // Pointer to VEM and specific data to be sent / Pointer to Specific data in VD local send DB
      ptrSpecDataVDCommLocalSndStruct AT ptrSpecDataVDCommLocalSnd : Struct   // Pointer to Specific data in VD local send DB - Structure
         ID : Byte;
         DataType : Byte;
         ReplicationFactor : Word;
         DbNbr : Word;
         CrossAreaPointer : DWord;
      END_STRUCT;
   END_VAR
   VAR CONSTANT
      SECTION_OUTPUTS : Bool := TRUE;   // Section - Outputs
      SECTION_HMI : Bool := TRUE;   // Section - HMI
      PART_LOST_DLY : DInt := 1000;
      VEM_DATA_OFFSET : DWord;
      SPEC_DATA_OFFSET : DWord := 16#100;
      VDCOM_DATA_OFFSET : DWord := 10;
      VDCOM_VEM_DATA_OFFSET : DWord := 10;
      VDCOM_SPEC_DATA_OFFSET : DWord := 266;
      DATA_TYPE_BYTE : Byte := 16#02;
      AREA_IDENTIFIER : DWord := 16#84000000;
      POINTER_SYNTAX_ID : Byte := 16#10;
      ON : Word := 16#0001;
      OFF : Word := 16#0000;
      DATA_SND_TIME_MAX : Time := T#10S;
      DATA_RCV_TIME_MAX : Time := T#15S;
      STAT_CODE_BUSY : Int := 2;   // Status code - job busy
      STAT_CODE_SUCCESS : Int := 1;   // Status code - job successful
      STAT_CODE_SND_FINISH_NOK : Int := -3;   // Status code - No Send finished
      STAT_CODE_START_WITHOUT_ID : Int := -4;   // Status code - ID not valid or missing
      STAT_CODE_RCV_DATA_NOK : Int := -5;   // Status code - Received data is NOK
      STAT_CODE_RCV_NEW_DATA_OVTIME : Int := -9;   // Status code - New Data Received Overtime
      CMD_GET_VEM_DATA : DWord := 1002;
      SPECIFIC_DATA_LENGTH_MAX : DInt := 7026;
      STATUS_001 : Int := 1;   // Status - 001 : Success
      STATUS_MINUS_003 : Int := -3;   // Status - 003 : Error sending message to virtual device
      STATUS_MINUS_006 : Int := -6;   // Status - 006 : Error ID not valid or missing
      STATUS_MINUS_001 : Int := -1;   // Status - 001 :
      STATUS_MINUS_005 : Int := -5;   // Status -009 : Error no response received from virtual device
      STATUS_MINUS_009 : Int := -9;   // Status -009 : Error no response received from virtual device
      VISIBLE : Word := 16#0001;   // Enable
      ENABLE : Word := 16#0002;   // Visible
      COLOUR_DEFAULT : Word := 16#0000;   // Colour - Default
      COLOUR_RED : Word := 16#0010;   // Colour - Red
      COLOUR_GREEN : Word := 16#0020;   // Colour - Green
      COLOUR_BLUE : Word := 16#0040;   // Colour - Blue
      COLOUR_WHITE : Word := 16#0080;   // Colour - White
      COLOUR_BLUE_FLASH : Word := 16#0400;   // Colour - Blue flash
   END_VAR
BEGIN
   (******************************************************************************
    Changelog

       17W24D4 10:00H PMo
       - Section outputs is now true

       17W23D5 17:00H PMo
       - Conversion from FBD TO SCL

       18W3D5 : AHE
       - Confirm.ok.begin will not clear VEM data

    19W12D4 : WDL
       - Decoding of BodyTypeMatrix removed

    List OF authors

       Company : Volvo Cars Gent
       Name    : Patrick Moreau (PMo)
       E-mail  : patrick.moreau@volvocars.com
       Tel.    : +32 9 2503165

    Description

       This module is part OF the VIDS suite AND is the principal module TO be
       integrated FOR RFID, Track, Confirm AND other submodules.
       Its main purpose is TO communicate with the production servers via virtual
       device AND retrieve VEM data OR specific data 

    ******************************************************************************)

   (******************************************************************************)
   (* Create pointers                                                            *)
   (******************************************************************************)

   //Copy pointers
   #ptrIO_VEMData := #IO_VEMData;
   #ptrIO_VEMDataChange := #IO_VEMDataChange;
   #ptrIO_SpecData := #IO_SpecificData;

   //Create pointer to VEMData in VDComm local receive DB
   #ptrVEMDataVDCommLocalRcvStruct.ID := #POINTER_SYNTAX_ID;
   #ptrVEMDataVDCommLocalRcvStruct.DataType := #DATA_TYPE_BYTE;
   #ptrVEMDataVDCommLocalRcvStruct.ReplicationFactor := 256;
   #ptrVEMDataVDCommLocalRcvStruct.DbNbr := UINT_TO_WORD(DB_ANY_TO_UINT(#C_VDCommLocalRcvDB));
   #ptrVEMDataVDCommLocalRcvStruct.CrossAreaPointer := SHL(IN := #VDCOM_VEM_DATA_OFFSET, N := 3) OR #AREA_IDENTIFIER; //Offset 10

   //Create pointer to Specific data in VDComm local receive DB
   #ptrSpecDataVDCommLocalRcvStruct.ID := #POINTER_SYNTAX_ID;
   #ptrSpecDataVDCommLocalRcvStruct.DataType := #DATA_TYPE_BYTE;
   #ptrSpecDataVDCommLocalRcvStruct.ReplicationFactor := 7026;
   #ptrSpecDataVDCommLocalRcvStruct.DbNbr := UINT_TO_WORD(DB_ANY_TO_UINT(#C_VDCommLocalRcvDB));
   #ptrSpecDataVDCommLocalRcvStruct.CrossAreaPointer := SHL(IN := #VDCOM_SPEC_DATA_OFFSET, N := 3) OR #AREA_IDENTIFIER; //Offset 266

   //Create pointer to VEMData in VDComm local send DB
   #ptrVEMDataVDCommLocalSndStruct.ID := #POINTER_SYNTAX_ID;
   #ptrVEMDataVDCommLocalSndStruct.DataType := #DATA_TYPE_BYTE;
   #ptrVEMDataVDCommLocalSndStruct.ReplicationFactor := 256;
   #ptrVEMDataVDCommLocalSndStruct.DbNbr := UINT_TO_WORD(DB_ANY_TO_UINT(#C_VDCommLocalSndDB));
   #ptrVEMDataVDCommLocalSndStruct.CrossAreaPointer := SHL(IN := #VDCOM_VEM_DATA_OFFSET, N := 3) OR #AREA_IDENTIFIER; //Offset 10

   //Create pointer to Specific data in VDComm local send DB
   #ptrSpecDataVDCommLocalSndStruct.ID := #POINTER_SYNTAX_ID;
   #ptrSpecDataVDCommLocalSndStruct.DataType := #DATA_TYPE_BYTE;
   #ptrSpecDataVDCommLocalSndStruct.ReplicationFactor := 2048;
   #ptrSpecDataVDCommLocalSndStruct.DbNbr := UINT_TO_WORD(DB_ANY_TO_UINT(#C_VDCommLocalSndDB));
   #ptrSpecDataVDCommLocalSndStruct.CrossAreaPointer := SHL(IN := #VDCOM_SPEC_DATA_OFFSET, N := 3) OR #AREA_IDENTIFIER; //Offset 266

   (******************************************************************************)
   (* Inputs                                                                     *)
   (******************************************************************************)

   #_PartLostDlyTmr(I_StartTimer:=#PartPres AND NOT #I_PartPres,
                 I_HoldTimer:=FALSE,
                 I_MaxTimerValue:=#PART_LOST_DLY,
                 O_TimerResult=>#PartLostDlyTmrElapsed,
                 O_TimerValue=>#PartLostDlyTmrAct);

   #PartPres := #I_PartPres OR #PartPres AND NOT #PartLostDlyTmrElapsed;

   (******************************************************************************)
   (* Create pulses                                                              *)
   (******************************************************************************)

   //Get VEM Data - Create start pulse
   #StartGetVEMDataPls := #I_StartGetVEMData AND NOT #StartGetVEMDataEdg;
   #StartGetVEMDataEdg := #I_StartGetVEMData;

   //Create pulse on part lost
   #PartLostPls := NOT #IO_VIDS.PartPres AND #PartLostEdg;
   #PartLostEdg := #IO_VIDS.PartPres;

   (******************************************************************************)
   (* Initialize all                                                             *)
   (******************************************************************************)

   IF #PartLostPls THEN

       #RetVal := FILL(BVAL := #EmptyByte, BLK => #VEMDataInitArray);  //Create init array
       #StepNbr := 0;                                                  //Reset sequence
       #VEMDataValid := FALSE;                                 //Reset VEM data valid
       #VEMDataNotValid := FALSE;                              //Reset VEM data not valid
       #Status := 0;                                                   //Reset status

       //Initialize IO_VIDS.VEMData
       #DeserializePos := 0;
       #RetVal := Deserialize(SRC_ARRAY := #VEMDataInitArray, DEST_VARIABLE => #IO_VIDS.VEMData, POS := #DeserializePos);
       #RetVal := FILL(BVAL := #SPACE, BLK => #IO_VIDS.VEMData.UserID);
       #RetVal := FILL(BVAL := #SPACE, BLK => #IO_VIDS.VEMData.Variant);
       #RetVal := FILL(BVAL := #SPACE, BLK => #IO_VIDS.VEMData.VinNumber);
       #RetVal := FILL(BVAL := #SPACE, BLK => #IO_VIDS.VEMData.PopIDSuffix);

       //Initialize IO_VIDS.Specific data
       #RetVal := FILL(BVAL := #EmptyByte, BLK => #IO_VIDS.SpecificDataInit);

       //Initialize IO_VEMData
       #DeserializePos := 0;
       #RetVal:=Deserialize(SRC_ARRAY := #VEMDataInitArray, DEST_VARIABLE => #IO_VEMData, POS := #DeserializePos);
       #RetVal := FILL(BVAL := #SPACE, BLK => #IO_VEMData.UserID);
       #RetVal := FILL(BVAL := #SPACE, BLK => #IO_VEMData.Variant);
       #RetVal := FILL(BVAL := #SPACE, BLK => #IO_VEMData.VinNumber);
       #RetVal := FILL(BVAL := #SPACE, BLK => #IO_VEMData.PopIDSuffix);

       //Initialize IO_Specific data
       #RetVal := FILL(BVAL := #EmptyByte, BLK => #IO_SpecificData);

       //Initialize IO_VEMDataChange
       #DeserializePos := 0;
       #RetVal := Deserialize(SRC_ARRAY := #VEMDataInitArray, DEST_VARIABLE => #IO_VEMDataChange, POS := #DeserializePos);
       #RetVal := FILL(BVAL := #SPACE, BLK => #IO_VEMDataChange.UserID);
       #RetVal := FILL(BVAL := #SPACE, BLK => #IO_VEMDataChange.Variant);
       #RetVal := FILL(BVAL := #SPACE, BLK => #IO_VEMDataChange.VinNumber);
       #RetVal := FILL(BVAL := #SPACE, BLK => #IO_VEMDataChange.PopIDSuffix);

       //Reset signals
       #IO_VIDS.GetVEMData.BeginReqMem := FALSE;
       #IO_VIDS.GetVEMData.Running := FALSE;

       #IO_VIDS.ChangeData.BeginReqMem := FALSE;
       #IO_VIDS.ChangeData.Running := FALSE;

       #IO_VIDS.InitTag.BeginReqMem := FALSE;
       #IO_VIDS.InitTag.Running := FALSE;

       #IO_VIDS.GetVEMDataByRFID.BeginReqMem := FALSE;
       #IO_VIDS.GetVEMDataByRFID.Running := FALSE;

       #IO_VIDS.ReplaceTag.BeginReqMem := FALSE;
       #IO_VIDS.ReplaceTag.Running := FALSE;

       #IO_VIDS.Confirm.BeginReqMem := FALSE;
       #IO_VIDS.Confirm.Running := FALSE;

       #IO_VIDS.Track.BeginReqMem := FALSE;
       #IO_VIDS.Track.Running := FALSE;

       #IO_VIDS.Couple.BeginReqMem := FALSE;
       #IO_VIDS.Couple.Running := FALSE;

       #IO_VIDS.DeCouple.BeginReqMem := FALSE;
       #IO_VIDS.DeCouple.Running := FALSE;

       #IO_VIDS.GetNextID.BeginReqMem := FALSE;
       #IO_VIDS.GetNextID.Running := FALSE;

       #IO_VIDS.GetSpecData.BeginReqMem := FALSE;
       #IO_VIDS.GetSpecData.Running := FALSE;

       #IO_VIDS.PutSpecData.BeginReqMem := FALSE;
       #IO_VIDS.PutSpecData.Running := FALSE;

   END_IF;

   //Running summary
   #Busy :=
   #IO_VIDS.GetVEMData.Running OR
   #IO_VIDS.ChangeData.Running OR
   #IO_VIDS.InitTag.Running OR
   #IO_VIDS.GetVEMDataByRFID.Running OR
   #IO_VIDS.ReplaceTag.Running OR
   #IO_VIDS.Track.Running OR
   #IO_VIDS.Confirm.Running OR
   #IO_VIDS.Couple.Running OR
   #IO_VIDS.DeCouple.Running OR
   #IO_VIDS.GetNextID.Running OR
   #IO_VIDS.GetSpecData.Running OR
   #IO_VIDS.PutSpecData.Running;

   (******************************************************************************)
   (* Get VEM data                                                               *)
   (******************************************************************************)

   //Get VEM Data - Begin request
   #IO_VIDS.GetVEMData.BeginReq := #StartGetVEMDataPls;

   //Get VEM data - Memorize parameters
   IF #IO_VIDS.GetVEMData.BeginReq THEN
       #TagIDMem := #I_TagID;
       #BodyIDMem := #I_BodyID;
       #CarrierIDMem := #I_CarrierID;
       #MixNbrMem := #I_MixNbr;
       #PopIDMem := #I_PopID;
       #PopIDSuffixMem := #I_PopIDSuffix;
       #PopTypeMem := #I_PopType;

   END_IF;

   //Get VEM data - Initialize parameters
   IF #IO_VIDS.GetVEMData.OkBegin THEN

       #IO_VIDS.VEMData.CommandCode := #CMD_GET_VEM_DATA;
       #IO_VIDS.VEMData.Identification := #TagIDMem;
       #IO_VIDS.VEMData.BodyID := #BodyIDMem;
       #IO_VIDS.VEMData.CarrierID := #CarrierIDMem;
       #IO_VIDS.VEMData.MixNumber := #MixNbrMem;
       #IO_VIDS.VEMData.IdType := #C_IDType;
       #IO_VIDS.VEMData.PopID := #PopIDMem;
       #IO_VIDS.VEMData.PopIDSuffix := #PopIDSuffixMem;
       #IO_VIDS.VEMData.PopType := #PopTypeMem;
   END_IF;

   //Get VEM data - Begin
   #IO_VIDS.GetVEMData.Begin := #IO_VIDS.GetVEMData.OkBegin;

   //Get VEM Data - Busy
   #BusyGetVEMData := #IO_VIDS.GetVEMData.Running;

   (******************************************************************************)
   (* Memorize begin request                                                     *)
   (******************************************************************************)

   //Get VEM Data - Memorize begin request
   IF #IO_VIDS.GetVEMData.BeginReq AND NOT #GetVEMDataBeginReqEdg THEN
       #IO_VIDS.GetVEMData.BeginReqMem := TRUE;
   END_IF;
   #GetVEMDataBeginReqEdg := #IO_VIDS.GetVEMData.BeginReq;

   //Change VEM Data - Memorize begin request
   IF #IO_VIDS.ChangeData.BeginReq AND NOT #ChangeDataBeginReqEdg THEN
       #IO_VIDS.ChangeData.BeginReqMem := TRUE;
   END_IF;
   #ChangeDataBeginReqEdg := #IO_VIDS.ChangeData.BeginReq;

   //Init tag - Memorize begin request
   IF #IO_VIDS.InitTag.BeginReq AND NOT #InitTagBeginReqEdg THEN
       #IO_VIDS.InitTag.BeginReqMem := TRUE;
   END_IF;
   #InitTagBeginReqEdg := #IO_VIDS.InitTag.BeginReq;

   //Get VEM Data by RFID - Memorize begin request
   IF #IO_VIDS.GetVEMDataByRFID.BeginReq AND NOT #GetVEMDataByRFIDBeginReqEdg THEN
       #IO_VIDS.GetVEMDataByRFID.BeginReqMem := TRUE;
   END_IF;
   #GetVEMDataByRFIDBeginReqEdg := #IO_VIDS.GetVEMDataByRFID.BeginReq;

   //Replace tag - Memorize begin request
   IF #IO_VIDS.ReplaceTag.BeginReq AND NOT #ReplaceTagBeginReqEdg THEN
       #IO_VIDS.ReplaceTag.BeginReqMem := TRUE;
   END_IF;
   #ReplaceTagBeginReqEdg := #IO_VIDS.ReplaceTag.BeginReq;

   //Track - Memorize begin request
   IF #IO_VIDS.Track.BeginReq AND NOT #TrackBeginReqEdg THEN
       #IO_VIDS.Track.BeginReqMem := TRUE;
   END_IF;
   #TrackBeginReqEdg := #IO_VIDS.Track.BeginReq;

   //Confirm - Memorize begin request
   IF #IO_VIDS.Confirm.BeginReq AND NOT #ConfirmBeginReqEdg THEN
       #IO_VIDS.Confirm.BeginReqMem := TRUE;
   END_IF;
   #ConfirmBeginReqEdg := #IO_VIDS.Confirm.BeginReq;

   //Couple - Memorize begin request
   IF #IO_VIDS.Couple.BeginReq AND NOT #CoupleBeginReqEdg THEN
       #IO_VIDS.Couple.BeginReqMem := TRUE;
   END_IF;
   #CoupleBeginReqEdg := #IO_VIDS.Couple.BeginReq;

   //Decouple - Memorize begin request
   IF #IO_VIDS.DeCouple.BeginReq AND NOT #DecoupleBeginReqEdg THEN
       #IO_VIDS.DeCouple.BeginReqMem := TRUE;
   END_IF;
   #DecoupleBeginReqEdg := #IO_VIDS.DeCouple.BeginReq;

   //Get next ID - Memorize begin request
   IF #IO_VIDS.GetNextID.BeginReq AND NOT #GetNextIDBeginReqEdg THEN
       #IO_VIDS.GetNextID.BeginReqMem := TRUE;
   END_IF;
   #GetNextIDBeginReqEdg := #IO_VIDS.GetNextID.BeginReq;

   //Get Specific data - Memorize begin request
   IF #IO_VIDS.GetSpecData.BeginReq AND NOT #GetSpecDataBeginReqEdg THEN
       #IO_VIDS.GetSpecData.BeginReqMem := TRUE;
   END_IF;
   #GetSpecDataBeginReqEdg := #IO_VIDS.GetSpecData.BeginReq;

   //Put specific data - Memorize begin request
   IF #IO_VIDS.PutSpecData.BeginReq AND NOT #PutSpecDataBeginReqEdg THEN
       #IO_VIDS.PutSpecData.BeginReqMem := TRUE;
   END_IF;
   #PutSpecDataBeginReqEdg := #IO_VIDS.PutSpecData.BeginReq;

   (******************************************************************************)
   (* Running                                                                    *)
   (******************************************************************************)

   IF #IO_VIDS.GetVEMData.OkBegin AND #IO_VIDS.GetVEMData.Begin THEN
       #IO_VIDS.GetVEMData.Running := TRUE;
   ELSIF #IO_VIDS.ChangeData.OkBegin AND #IO_VIDS.ChangeData.Begin THEN
       #IO_VIDS.ChangeData.Running := TRUE;
   ELSIF #IO_VIDS.InitTag.OkBegin AND #IO_VIDS.InitTag.Begin THEN
       #IO_VIDS.InitTag.Running := TRUE;
   ELSIF #IO_VIDS.GetVEMDataByRFID.OkBegin AND #IO_VIDS.GetVEMDataByRFID.Begin THEN
       #IO_VIDS.GetVEMDataByRFID.Running := TRUE;
   ELSIF #IO_VIDS.ReplaceTag.OkBegin AND #IO_VIDS.ReplaceTag.Begin THEN
       #IO_VIDS.ReplaceTag.Running := TRUE;
   ELSIF #IO_VIDS.Track.OkBegin AND #IO_VIDS.Track.Begin THEN
       #IO_VIDS.Track.Running := TRUE;
   ELSIF #IO_VIDS.Confirm.OkBegin AND #IO_VIDS.Confirm.Begin THEN
       #IO_VIDS.Confirm.Running := TRUE;
   ELSIF #IO_VIDS.Couple.OkBegin AND #IO_VIDS.Couple.Begin THEN
       #IO_VIDS.Couple.Running := TRUE;
   ELSIF #IO_VIDS.DeCouple.OkBegin AND #IO_VIDS.DeCouple.Begin THEN
       #IO_VIDS.DeCouple.Running := TRUE;
   ELSIF #IO_VIDS.GetNextID.OkBegin AND #IO_VIDS.GetNextID.Begin THEN
       #IO_VIDS.GetNextID.Running := TRUE;
   ELSIF #IO_VIDS.GetSpecData.OkBegin AND #IO_VIDS.GetSpecData.Begin THEN
       #IO_VIDS.GetSpecData.Running := TRUE;
   ELSIF #IO_VIDS.PutSpecData.OkBegin AND #IO_VIDS.PutSpecData.Begin THEN
       #IO_VIDS.PutSpecData.Running := TRUE;
   END_IF;

   (******************************************************************************)
   (* Update status                                                              *)
   (******************************************************************************)

   IF #StepNbr > 0 THEN
       IF #IO_VIDS.GetVEMData.Running THEN
           #IO_VIDS.GetVEMData.Status := #Status;
       ELSIF #IO_VIDS.ChangeData.Running THEN
           #IO_VIDS.ChangeData.Status := #Status;
       ELSIF #IO_VIDS.InitTag.Running THEN
           #IO_VIDS.InitTag.Status := #Status;
       ELSIF #IO_VIDS.GetVEMDataByRFID.Running THEN
           #IO_VIDS.GetVEMDataByRFID.Status := #Status;
       ELSIF #IO_VIDS.ReplaceTag.Running THEN
           #IO_VIDS.ReplaceTag.Status := #Status;
       ELSIF #IO_VIDS.Track.Running THEN
           #IO_VIDS.Track.Status := #Status;
       ELSIF #IO_VIDS.Confirm.Running THEN
           #IO_VIDS.Confirm.Status := #Status;
       ELSIF #IO_VIDS.Couple.Running THEN
           #IO_VIDS.Couple.Status := #Status;
       ELSIF #IO_VIDS.DeCouple.Running THEN
           #IO_VIDS.DeCouple.Status := #Status;
       ELSIF #IO_VIDS.GetNextID.Running THEN
           #IO_VIDS.GetNextID.Status := #Status;
       ELSIF #IO_VIDS.GetSpecData.Running THEN
           #IO_VIDS.GetSpecData.Status := #Status;
       ELSIF #IO_VIDS.PutSpecData.Running THEN
           #IO_VIDS.PutSpecData.Status := #Status;
       END_IF;
   END_IF;

   (******************************************************************************)
   (* Step 0                                                                     *)
   (******************************************************************************)

   //Step 0 On Active - Reset locked
   //IF #StepNbr = 0 THEN

   //END_IF;

   (******************************************************************************)
   (* Step 0 TO 50                                                               *)
   (******************************************************************************)

   //Step 0 to 50
   IF #Step0To50Cond THEN
       #StepNbr := 50;
       #Step50EntryPls := TRUE;
   ELSE
       #Step50EntryPls := FALSE;
   END_IF;

   //Step 0 to 50 - Condition
   #Step0To50Cond :=
   #StepNbr = 0 AND (
   #IO_VIDS.GetVEMData.BeginReqMem OR
   #IO_VIDS.ChangeData.BeginReqMem OR
   #IO_VIDS.InitTag.BeginReqMem OR
   #IO_VIDS.GetVEMDataByRFID.BeginReqMem OR
   #IO_VIDS.ReplaceTag.BeginReqMem OR
   #IO_VIDS.Track.BeginReqMem OR
   #IO_VIDS.Confirm.BeginReqMem OR
   #IO_VIDS.Couple.BeginReqMem OR
   #IO_VIDS.DeCouple.BeginReqMem OR
   #IO_VIDS.GetNextID.BeginReqMem OR
   #IO_VIDS.GetSpecData.BeginReqMem OR
   #IO_VIDS.PutSpecData.BeginReqMem);

   (******************************************************************************)
   (* Step 50                                                                    *)
   (******************************************************************************)

   //Step 50 On Entry
   IF #Step50EntryPls THEN

       //Ok Begin
       IF #IO_VIDS.GetVEMData.BeginReqMem  THEN
           #IO_VIDS.GetVEMData.OkBegin := TRUE;
           #IO_VIDS.GetVEMData.BeginReqMem := FALSE;
       ELSIF #IO_VIDS.ChangeData.BeginReqMem  THEN
           #IO_VIDS.ChangeData.OkBegin := TRUE;
           #IO_VIDS.ChangeData.BeginReqMem := FALSE;
       ELSIF #IO_VIDS.InitTag.BeginReqMem  THEN
           #IO_VIDS.InitTag.OkBegin := TRUE;
           #IO_VIDS.InitTag.BeginReqMem := FALSE;
       ELSIF #IO_VIDS.GetVEMDataByRFID.BeginReqMem  THEN
           #IO_VIDS.GetVEMDataByRFID.OkBegin := TRUE;
           #IO_VIDS.GetVEMDataByRFID.BeginReqMem := FALSE;
       ELSIF #IO_VIDS.ReplaceTag.BeginReqMem THEN
           #IO_VIDS.ReplaceTag.OkBegin := TRUE;
           #IO_VIDS.ReplaceTag.BeginReqMem := FALSE;
       ELSIF #IO_VIDS.Track.BeginReqMem  THEN
           #IO_VIDS.Track.OkBegin := TRUE;
           #IO_VIDS.Track.BeginReqMem := FALSE;
       ELSIF #IO_VIDS.Confirm.BeginReqMem  THEN
           #IO_VIDS.Confirm.OkBegin := TRUE;
           #IO_VIDS.Confirm.BeginReqMem := FALSE;
       ELSIF #IO_VIDS.Couple.BeginReqMem  THEN
           #IO_VIDS.Couple.OkBegin := TRUE;
           #IO_VIDS.Couple.BeginReqMem := FALSE;
       ELSIF #IO_VIDS.DeCouple.BeginReqMem THEN
           #IO_VIDS.DeCouple.OkBegin := TRUE;
           #IO_VIDS.DeCouple.BeginReqMem := FALSE;
       ELSIF #IO_VIDS.GetNextID.BeginReqMem THEN
           #IO_VIDS.GetNextID.OkBegin := TRUE;
           #IO_VIDS.GetNextID.BeginReqMem := FALSE;
       ELSIF #IO_VIDS.GetSpecData.BeginReqMem  THEN
           #IO_VIDS.GetSpecData.OkBegin := TRUE;
           #IO_VIDS.GetSpecData.BeginReqMem := FALSE;
       ELSIF #IO_VIDS.PutSpecData.BeginReqMem  THEN
           #IO_VIDS.PutSpecData.OkBegin := TRUE;
           #IO_VIDS.PutSpecData.BeginReqMem := FALSE;
       END_IF;

       //Initialize commands
       #CmdCodeSent := 0;
       #CmdCodeRcvd := 0;

       //Initialize
       IF NOT #IO_VIDS.Track.OkBegin  AND NOT #IO_VIDS.GetNextID.OkBegin AND NOT #IO_VIDS.Confirm.OkBegin THEN

           //Initialize IO_VIDS.VEMData
           #DeserializePos := 0;
           #RetVal := Deserialize(SRC_ARRAY := #VEMDataInitArray, DEST_VARIABLE => #IO_VIDS.VEMData, POS := #DeserializePos);
           #RetVal := FILL(BVAL := #SPACE, BLK => #IO_VIDS.VEMData.UserID);
           #RetVal := FILL(BVAL := #SPACE, BLK => #IO_VIDS.VEMData.Variant);
           #RetVal := FILL(BVAL := #SPACE, BLK => #IO_VIDS.VEMData.VinNumber);
           #RetVal := FILL(BVAL := #SPACE, BLK => #IO_VIDS.VEMData.PopIDSuffix);

           //Initialize IO_VIDS.Specific data
           #RetVal := FILL(BVAL := #EmptyByte, BLK => #IO_VIDS.SpecificDataInit);

           //Initialize IO_VEMData
           #DeserializePos := 0;
           #RetVal := Deserialize(SRC_ARRAY := #VEMDataInitArray, DEST_VARIABLE => #IO_VEMData, POS := #DeserializePos);
           #RetVal := FILL(BVAL := #SPACE, BLK => #IO_VEMData.UserID);
           #RetVal := FILL(BVAL := #SPACE, BLK => #IO_VEMData.Variant);
           #RetVal := FILL(BVAL := #SPACE, BLK => #IO_VEMData.VinNumber);
           #RetVal := FILL(BVAL := #SPACE, BLK => #IO_VEMData.PopIDSuffix);

           //Initialize IO_Specific data
           #RetVal := FILL(BVAL := #EmptyByte, BLK => #IO_SpecificData);

           //Reset validation
           #VEMDataValid := FALSE;
           #VEMDataNotValid := FALSE;

       END_IF;

   ELSE
       #IO_VIDS.GetVEMData.OkBegin := FALSE;
       #IO_VIDS.ChangeData.OkBegin := FALSE;
       #IO_VIDS.InitTag.OkBegin := FALSE;
       #IO_VIDS.GetVEMDataByRFID.OkBegin := FALSE;
       #IO_VIDS.ReplaceTag.OkBegin := FALSE;
       #IO_VIDS.Track.OkBegin := FALSE;
       #IO_VIDS.Confirm.OkBegin := FALSE;
       #IO_VIDS.Couple.OkBegin := FALSE;
       #IO_VIDS.DeCouple.OkBegin := FALSE;
       #IO_VIDS.GetNextID.OkBegin := FALSE;
       #IO_VIDS.GetSpecData.OkBegin := FALSE;
       #IO_VIDS.PutSpecData.OkBegin := FALSE;
       #OkBegin := False;

   END_IF;

   //Step 50 on Active - Step Timer - Start
   #_Step50Tmr(I_StartTimer:=#StepNbr=50,
               I_HoldTimer:=FALSE,
               I_MaxTimerValue:=5000,
               O_TimerResult=>#Step50TmrElapsed,
               O_TimerValue=>#Step50TmrAct);

   //Step 50 On Active - Step Timer - Error overtime
   IF #Step50TmrElapsed THEN
       #Status := #STAT_CODE_RCV_NEW_DATA_OVTIME;
   END_IF;

   //Step 50 On Active - Step Timer - Memorize maximum
   IF #Step50TmrAct > #Step50TmrActMax THEN
       #Step50TmrActMax := #Step50TmrAct;
   END_IF;

   (******************************************************************************)
   (* Step 50 TO 100                                                             *)
   (******************************************************************************)

   //Step 50 to 100
   IF #Step50To100Cond THEN
       #StepNbr := 100;
       #Step100EntryPls := TRUE;
   ELSE
       #Step100EntryPls := FALSE;
   END_IF;

   //Step 50 to 200
   IF #Step50To200Cond THEN
       #StepNbr := 200;
       #Step200EntryPls := TRUE;
   ELSE
       #Step200EntryPls := FALSE;
   END_IF;

   //Step 0 - Exit pulse
   #Step0ExitPls := #Step50EntryPls;

   //Step 50 to 100 - Condition
   #Step50To100Cond := #StepNbr = 50 AND #IO_VIDS.GetVEMDataByRFID.Running;

   //Step 50 TO 200 - Condition
   #Step50To200Cond:= #StepNbr=50 AND
   (#IO_VIDS.GetVEMData.Running OR
   #IO_VIDS.ChangeData.Running OR
   #IO_VIDS.InitTag.Running OR
   #IO_VIDS.ReplaceTag.Running OR
   #IO_VIDS.Track.Running OR
   #IO_VIDS.Confirm.Running OR
   #IO_VIDS.Couple.Running OR
   #IO_VIDS.DeCouple.Running OR
   #IO_VIDS.GetNextID.Running OR
   #IO_VIDS.GetSpecData.Running OR
   #IO_VIDS.PutSpecData.Running);

   (******************************************************************************)
   (* Step 100                                                                   *)
   (******************************************************************************)

   // Step 0 On Exit
   IF #Step0ExitPls THEN

       #Status := #STAT_CODE_BUSY; //Status busy

   END_IF;


   //Step 100 On Active - New data received
   IF #StepNbr = 100 AND #NewData THEN
       //Copy received VEM data
       #RetVal := BLKMOV(SRCBLK := #ptrVEMDataVDCommLocalRcv, DSTBLK => #VEMDataRcvArray);
       #DeserializePos := 0;
       #RetVal:=Deserialize(SRC_ARRAY := #VEMDataRcvArray, DEST_VARIABLE => #IO_VIDS.VEMData, POS := #DeserializePos);

       #CmdCodeRcvd := #IO_VIDS.VEMData.CommandCode;
       //Update #Status
       IF #IO_VIDS.VEMData.ErrorCode < 0 THEN
           #Status := DINT_TO_INT(#IO_VIDS.VEMData.ErrorCode);
       ELSE
           #IO_VEMData.Identification := #IO_VIDS.VEMData.Identification;
       END_IF;
   END_IF;

   //Step 100 on Active - Step Timer - Start
   #_Step100Tmr(I_StartTimer := #StepNbr = 100,
                I_HoldTimer := FALSE,
                I_MaxTimerValue := 15000,
                O_TimerResult => #Step100TmrElapsed,
                O_TimerValue => #Step100TmrAct);

   //Step 100 On Active - Step Timer - Error overtime
   IF #Step100TmrElapsed THEN
       #Status := #STAT_CODE_RCV_NEW_DATA_OVTIME;
   END_IF;

   //Step 100 On Active - Step Timer - Memorize maximum
   IF #Step100TmrAct > #Step100TmrActMax THEN
       #Step100TmrActMax := #Step100TmrAct;
   END_IF;

